// TIA Portal project "tictactoe_v2" (V14)

(* hardware
DEVICE "S7-1200 station_1"  S7-1200 Station
   slot 0: "Rack_0"  S7-1200 Rack  Rack  V1.0
   slot 1: "PLC_1"  CPU 1212C DC/DC/Rly  6ES7 212-1HE40-0XB0  V4.2
DEVICE "HMI_1"  KTP600 Basic color PN
   slot 0: "KTP600 Basic color PN"  KTP600 Basic color PN  6AV6 647-0AD11-3AX0  12.0.0.0
   slot 1: "HMI_RT_1"  KTP600 Basic color PN  6AV6 647-0AD11-3AX0  12.0.0.0
   slot 5: "HMI_1.IE_CP_1"  PROFINET Interface  12.0.0.0
      slot 1: "PROFINET Interface_1"  PROFINET Interface
         slot 1: "Port_1"  Port
*)

// ===== PLC "PLC_1"  CPU 1212C DC/DC/Rly =====

VAR_GLOBAL   // PLC tag table "Global"
   "x" AT %M15.2 : Bool;
   "Reset" AT %M12.1 : Bool;
   "GameType" AT %MB17 : SInt;
END_VAR

VAR_GLOBAL   // PLC tag table "3x3Tags"
   "t00" AT %MB1 : SInt;
   "t01" AT %MB2 : SInt;
   "t02" AT %MB3 : SInt;
   "t10" AT %MB4 : SInt;
   "t11" AT %MB10 : SInt;
   "t12" AT %MB13 : SInt;
   "t20" AT %MB7 : SInt;
   "t21" AT %MB8 : SInt;
   "t22" AT %MB9 : SInt;
   "t00btn" AT %M5.1 : Bool;
   "t01btn" AT %M5.2 : Bool;
   "t02btn" AT %M5.3 : Bool;
   "t10btn" AT %M5.4 : Bool;
   "t11btn" AT %M5.5 : Bool;
   "t12btn" AT %M5.6 : Bool;
   "t20btn" AT %M5.7 : Bool;
   "t21btn" AT %M6.0 : Bool;
   "t22btn" AT %M6.1 : Bool;
   "WinValue" AT %MB36 : SInt;
   "Stop" AT %M37.0 : Bool;
   "BotsTurn" AT %M37.1 : Bool;
   "t03" AT %MB46 : SInt;
   "t13" AT %MB38 : SInt;
   "t23" AT %MB39 : SInt;
   "t33" AT %MB40 : SInt;
   "t32" AT %MB41 : SInt;
   "t31" AT %MB42 : SInt;
   "t30" AT %MB43 : SInt;
   "t03btn" AT %M44.0 : Bool;
   "t13btn" AT %M44.1 : Bool;
   "t23btn" AT %M44.2 : Bool;
   "t33btn" AT %M44.3 : Bool;
   "t32btn" AT %M44.4 : Bool;
   "t31btn" AT %M44.5 : Bool;
   "t30btn" AT %M44.6 : Bool;
END_VAR

FUNCTION "ResetAllVariables" : Void   // FC1, LAD
{ S7_Optimized_Access := 'TRUE' }
VERSION : 0.1
BEGIN

REGION Network 1
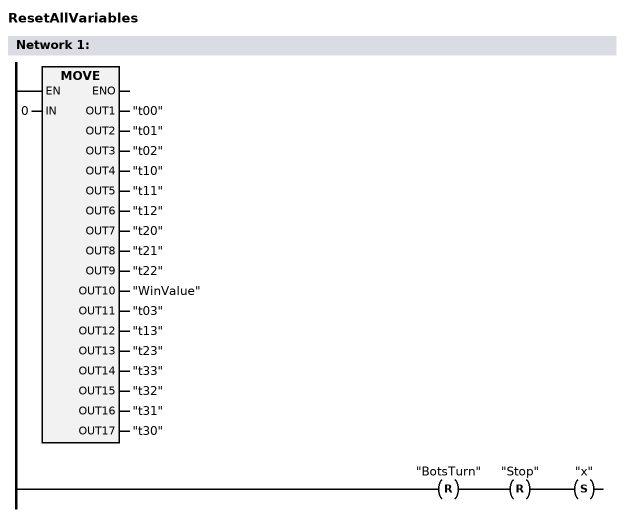
   RUNG wire#powerrail
      Move(in := 0, out1 => "t00", out2 => "t01", out3 => "t02", out4 => "t10", out5 => "t11", out6 => "t12", out7 => "t20", out8 => "t21", out9 => "t22", out10 => "WinValue", out11 => "t03", out12 => "t13", out13 => "t23", out14 => "t33", out15 => "t32", out16 => "t31", out17 => "t30")
   END_RUNG
   RUNG wire#powerrail
      R_Coil( "BotsTurn" )
      R_Coil( "Stop" )
      S_Coil( "x" )
   END_RUNG
   // the same network as SCL:
   "t00" := 0;
   "t01" := 0;
   "t02" := 0;
   "t10" := 0;
   "t11" := 0;
   "t12" := 0;
   "t20" := 0;
   "t21" := 0;
   "t22" := 0;
   "WinValue" := 0;
   "t03" := 0;
   "t13" := 0;
   "t23" := 0;
   "t33" := 0;
   "t32" := 0;
   "t31" := 0;
   "t30" := 0;
   "BotsTurn" := FALSE;
   "Stop" := FALSE;
   "x" := TRUE;
END_REGION
END_FUNCTION

FUNCTION "ChangeXValue" : Void   // FC4, LAD
{ S7_Optimized_Access := 'TRUE' }
VERSION : 0.1
   VAR_INPUT
      x : Bool;
   END_VAR
   VAR_OUTPUT
      value : Int;
   END_VAR
BEGIN

REGION Network 1
   // W zależności od wartości zmiennej "x" zmiana zapisywanego "symbolu"
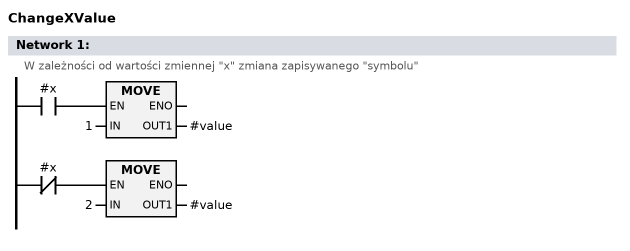
   RUNG wire#powerrail
      Contact( #x )
      Move(in := 1, out1 => #value)
   END_RUNG
   RUNG wire#powerrail
      I_Contact( #x )
      Move(in := 2, out1 => #value)
   END_RUNG
   // the same network as SCL:
   IF #x THEN #value := 1; END_IF;
   IF NOT #x THEN #value := 2; END_IF;
END_REGION
END_FUNCTION

ORGANIZATION_BLOCK "Main"   // OB1, LAD, ProgramCycle
TITLE = "Main Program Sweep (Cycle)"
{ S7_Optimized_Access := 'TRUE' }
VERSION : 0.1
   VAR_INPUT
      Initial_Call : Bool;   // Initial call of this OB
      Remanence : Bool;   // =True, if remanent data are available
   END_VAR
   VAR_TEMP
      temp : Bool;
      temp2 : Bool;
   END_VAR
BEGIN

REGION Network 1
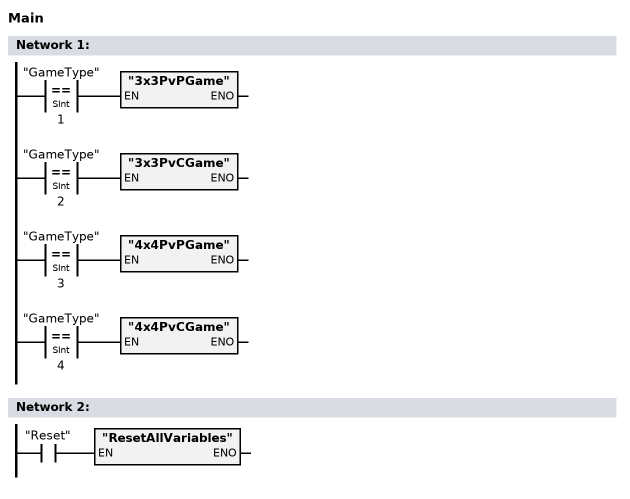
   RUNG wire#powerrail
      { S7_Templates := "SrcType := SInt" } EQ_Contact(in1 := "GameType", in2 := 1)
      "3x3PvPGame"()
   END_RUNG
   RUNG wire#powerrail
      { S7_Templates := "SrcType := SInt" } EQ_Contact(in1 := "GameType", in2 := 2)
      "3x3PvCGame"()
   END_RUNG
   RUNG wire#powerrail
      { S7_Templates := "SrcType := SInt" } EQ_Contact(in1 := "GameType", in2 := 3)
      "4x4PvPGame"()
   END_RUNG
   RUNG wire#powerrail
      { S7_Templates := "SrcType := SInt" } EQ_Contact(in1 := "GameType", in2 := 4)
      "4x4PvCGame"()
   END_RUNG
   // the same network as SCL:
   IF "GameType" = 1 THEN "3x3PvPGame"(); END_IF;
   IF "GameType" = 2 THEN "3x3PvCGame"(); END_IF;
   IF "GameType" = 3 THEN "4x4PvPGame"(); END_IF;
   IF "GameType" = 4 THEN "4x4PvCGame"(); END_IF;
END_REGION

REGION Network 2
   RUNG wire#powerrail
      Contact( "Reset" )
      "ResetAllVariables"()
   END_RUNG
   // the same network as SCL:
   IF "Reset" THEN "ResetAllVariables"(); END_IF;
END_REGION
END_ORGANIZATION_BLOCK

// folder: 3x3

FUNCTION "Check3x3" : Void   // FC2, LAD
{ S7_Optimized_Access := 'TRUE' }
VERSION : 0.1
   VAR_OUTPUT
      Stop : Bool;
      WinValue : SInt;
   END_VAR
BEGIN

REGION Network 1
   // Remis / X won!
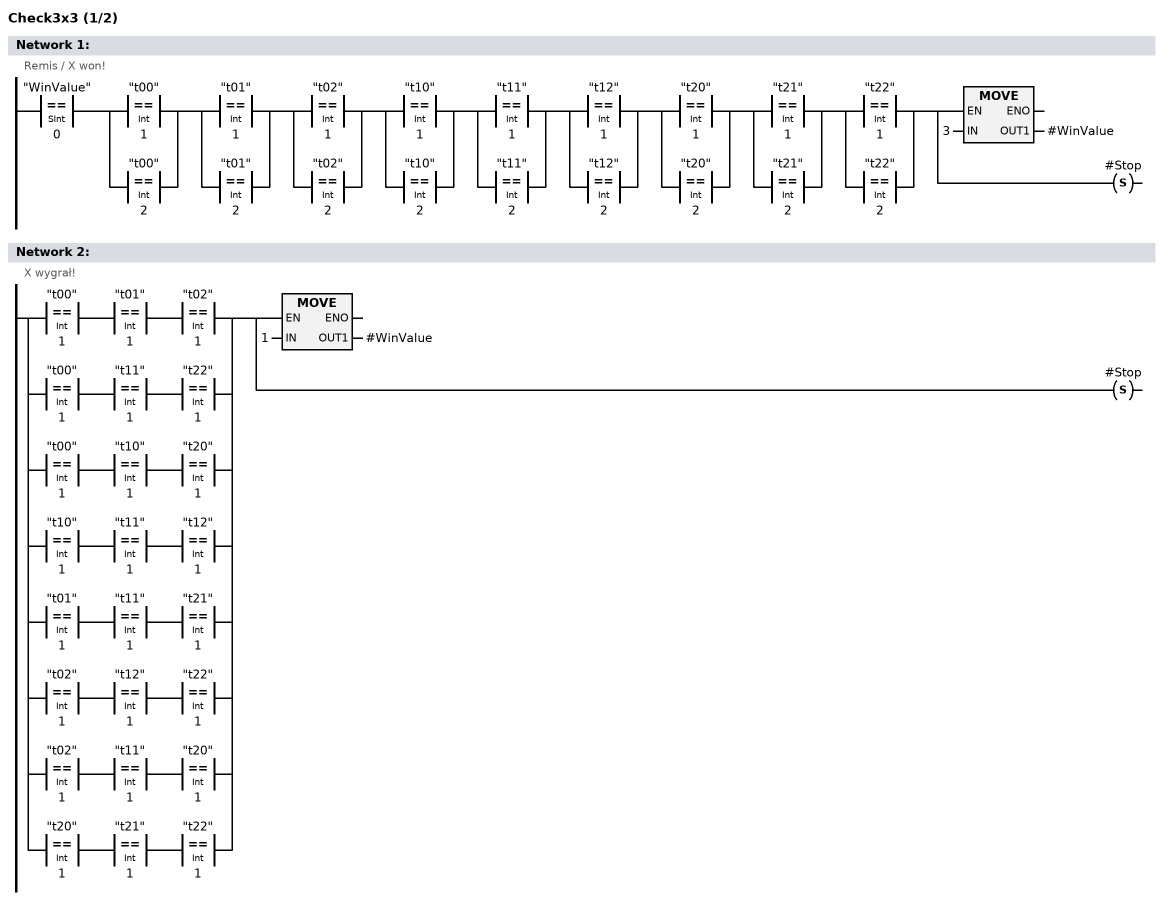
   RUNG wire#powerrail
      { S7_Templates := "SrcType := SInt" } EQ_Contact(in1 := "WinValue", in2 := 0)
      wire#w1
      { S7_Templates := "SrcType := Int" } EQ_Contact(in1 := "t00", in2 := 1)
      wire#w2
      { S7_Templates := "SrcType := Int" } EQ_Contact(in1 := "t01", in2 := 1)
      wire#w3
      { S7_Templates := "SrcType := Int" } EQ_Contact(in1 := "t02", in2 := 1)
      wire#w4
      { S7_Templates := "SrcType := Int" } EQ_Contact(in1 := "t10", in2 := 1)
      wire#w5
      { S7_Templates := "SrcType := Int" } EQ_Contact(in1 := "t11", in2 := 1)
      wire#w6
      { S7_Templates := "SrcType := Int" } EQ_Contact(in1 := "t12", in2 := 1)
      wire#w7
      { S7_Templates := "SrcType := Int" } EQ_Contact(in1 := "t20", in2 := 1)
      wire#w8
      { S7_Templates := "SrcType := Int" } EQ_Contact(in1 := "t21", in2 := 1)
      wire#w9
      { S7_Templates := "SrcType := Int" } EQ_Contact(in1 := "t22", in2 := 1)
      wire#w10
      Move(in := 3, out1 => #WinValue)
   END_RUNG
   RUNG wire#w1
      { S7_Templates := "SrcType := Int" } EQ_Contact(in1 := "t00", in2 := 2)
   END_RUNG wire#w2
   RUNG wire#w2
      { S7_Templates := "SrcType := Int" } EQ_Contact(in1 := "t01", in2 := 2)
   END_RUNG wire#w3
   RUNG wire#w3
      { S7_Templates := "SrcType := Int" } EQ_Contact(in1 := "t02", in2 := 2)
   END_RUNG wire#w4
   RUNG wire#w4
      { S7_Templates := "SrcType := Int" } EQ_Contact(in1 := "t10", in2 := 2)
   END_RUNG wire#w5
   RUNG wire#w5
      { S7_Templates := "SrcType := Int" } EQ_Contact(in1 := "t11", in2 := 2)
   END_RUNG wire#w6
   RUNG wire#w6
      { S7_Templates := "SrcType := Int" } EQ_Contact(in1 := "t12", in2 := 2)
   END_RUNG wire#w7
   RUNG wire#w7
      { S7_Templates := "SrcType := Int" } EQ_Contact(in1 := "t20", in2 := 2)
   END_RUNG wire#w8
   RUNG wire#w8
      { S7_Templates := "SrcType := Int" } EQ_Contact(in1 := "t21", in2 := 2)
   END_RUNG wire#w9
   RUNG wire#w9
      { S7_Templates := "SrcType := Int" } EQ_Contact(in1 := "t22", in2 := 2)
   END_RUNG wire#w10
   RUNG wire#w10
      S_Coil( #Stop )
   END_RUNG
   // the same network as SCL:
   IF ("WinValue" = 0) AND (("t00" = 1) OR ("t00" = 2)) AND (("t01" = 1) OR ("t01" = 2)) AND (("t02" = 1) OR ("t02" = 2)) AND (("t10" = 1) OR ("t10" = 2)) AND (("t11" = 1) OR ("t11" = 2)) AND (("t12" = 1) OR ("t12" = 2)) AND (("t20" = 1) OR ("t20" = 2)) AND (("t21" = 1) OR ("t21" = 2)) AND (("t22" = 1) OR ("t22" = 2)) THEN
       #WinValue := 3;
       #Stop := TRUE;
   END_IF;
END_REGION

REGION Network 2
   // X wygrał!
   RUNG wire#powerrail
      { S7_Templates := "SrcType := Int" } EQ_Contact(in1 := "t00", in2 := 1)
      { S7_Templates := "SrcType := Int" } EQ_Contact(in1 := "t01", in2 := 1)
      { S7_Templates := "SrcType := Int" } EQ_Contact(in1 := "t02", in2 := 1)
      wire#w1
      Move(in := 1, out1 => #WinValue)
   END_RUNG
   RUNG wire#powerrail
      { S7_Templates := "SrcType := Int" } EQ_Contact(in1 := "t00", in2 := 1)
      { S7_Templates := "SrcType := Int" } EQ_Contact(in1 := "t11", in2 := 1)
      { S7_Templates := "SrcType := Int" } EQ_Contact(in1 := "t22", in2 := 1)
   END_RUNG wire#w1
   RUNG wire#powerrail
      { S7_Templates := "SrcType := Int" } EQ_Contact(in1 := "t00", in2 := 1)
      { S7_Templates := "SrcType := Int" } EQ_Contact(in1 := "t10", in2 := 1)
      { S7_Templates := "SrcType := Int" } EQ_Contact(in1 := "t20", in2 := 1)
   END_RUNG wire#w1
   RUNG wire#powerrail
      { S7_Templates := "SrcType := Int" } EQ_Contact(in1 := "t10", in2 := 1)
      { S7_Templates := "SrcType := Int" } EQ_Contact(in1 := "t11", in2 := 1)
      { S7_Templates := "SrcType := Int" } EQ_Contact(in1 := "t12", in2 := 1)
   END_RUNG wire#w1
   RUNG wire#powerrail
      { S7_Templates := "SrcType := Int" } EQ_Contact(in1 := "t01", in2 := 1)
      { S7_Templates := "SrcType := Int" } EQ_Contact(in1 := "t11", in2 := 1)
      { S7_Templates := "SrcType := Int" } EQ_Contact(in1 := "t21", in2 := 1)
   END_RUNG wire#w1
   RUNG wire#powerrail
      { S7_Templates := "SrcType := Int" } EQ_Contact(in1 := "t02", in2 := 1)
      { S7_Templates := "SrcType := Int" } EQ_Contact(in1 := "t12", in2 := 1)
      { S7_Templates := "SrcType := Int" } EQ_Contact(in1 := "t22", in2 := 1)
   END_RUNG wire#w1
   RUNG wire#powerrail
      { S7_Templates := "SrcType := Int" } EQ_Contact(in1 := "t02", in2 := 1)
      { S7_Templates := "SrcType := Int" } EQ_Contact(in1 := "t11", in2 := 1)
      { S7_Templates := "SrcType := Int" } EQ_Contact(in1 := "t20", in2 := 1)
   END_RUNG wire#w1
   RUNG wire#powerrail
      { S7_Templates := "SrcType := Int" } EQ_Contact(in1 := "t20", in2 := 1)
      { S7_Templates := "SrcType := Int" } EQ_Contact(in1 := "t21", in2 := 1)
      { S7_Templates := "SrcType := Int" } EQ_Contact(in1 := "t22", in2 := 1)
   END_RUNG wire#w1
   RUNG wire#w1
      S_Coil( #Stop )
   END_RUNG
   // the same network as SCL:
   IF (("t00" = 1) AND ("t01" = 1) AND ("t02" = 1)) OR (("t00" = 1) AND ("t11" = 1) AND ("t22" = 1)) OR (("t00" = 1) AND ("t10" = 1) AND ("t20" = 1)) OR (("t10" = 1) AND ("t11" = 1) AND ("t12" = 1)) OR (("t01" = 1) AND ("t11" = 1) AND ("t21" = 1)) OR (("t02" = 1) AND ("t12" = 1) AND ("t22" = 1)) OR (("t02" = 1) AND ("t11" = 1) AND ("t20" = 1)) OR (("t20" = 1) AND ("t21" = 1) AND ("t22" = 1)) THEN
       #WinValue := 1;
       #Stop := TRUE;
   END_IF;
END_REGION

REGION Network 3
   // O wygrało! / O won! / O gewonnen!
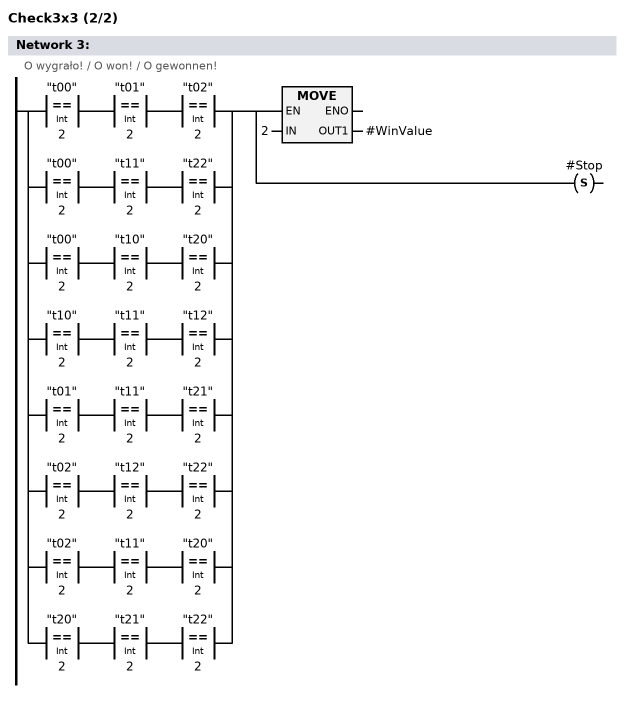
   RUNG wire#powerrail
      { S7_Templates := "SrcType := Int" } EQ_Contact(in1 := "t00", in2 := 2)
      { S7_Templates := "SrcType := Int" } EQ_Contact(in1 := "t01", in2 := 2)
      { S7_Templates := "SrcType := Int" } EQ_Contact(in1 := "t02", in2 := 2)
      wire#w1
      Move(in := 2, out1 => #WinValue)
   END_RUNG
   RUNG wire#powerrail
      { S7_Templates := "SrcType := Int" } EQ_Contact(in1 := "t00", in2 := 2)
      { S7_Templates := "SrcType := Int" } EQ_Contact(in1 := "t11", in2 := 2)
      { S7_Templates := "SrcType := Int" } EQ_Contact(in1 := "t22", in2 := 2)
   END_RUNG wire#w1
   RUNG wire#powerrail
      { S7_Templates := "SrcType := Int" } EQ_Contact(in1 := "t00", in2 := 2)
      { S7_Templates := "SrcType := Int" } EQ_Contact(in1 := "t10", in2 := 2)
      { S7_Templates := "SrcType := Int" } EQ_Contact(in1 := "t20", in2 := 2)
   END_RUNG wire#w1
   RUNG wire#powerrail
      { S7_Templates := "SrcType := Int" } EQ_Contact(in1 := "t10", in2 := 2)
      { S7_Templates := "SrcType := Int" } EQ_Contact(in1 := "t11", in2 := 2)
      { S7_Templates := "SrcType := Int" } EQ_Contact(in1 := "t12", in2 := 2)
   END_RUNG wire#w1
   RUNG wire#powerrail
      { S7_Templates := "SrcType := Int" } EQ_Contact(in1 := "t01", in2 := 2)
      { S7_Templates := "SrcType := Int" } EQ_Contact(in1 := "t11", in2 := 2)
      { S7_Templates := "SrcType := Int" } EQ_Contact(in1 := "t21", in2 := 2)
   END_RUNG wire#w1
   RUNG wire#powerrail
      { S7_Templates := "SrcType := Int" } EQ_Contact(in1 := "t02", in2 := 2)
      { S7_Templates := "SrcType := Int" } EQ_Contact(in1 := "t12", in2 := 2)
      { S7_Templates := "SrcType := Int" } EQ_Contact(in1 := "t22", in2 := 2)
   END_RUNG wire#w1
   RUNG wire#powerrail
      { S7_Templates := "SrcType := Int" } EQ_Contact(in1 := "t02", in2 := 2)
      { S7_Templates := "SrcType := Int" } EQ_Contact(in1 := "t11", in2 := 2)
      { S7_Templates := "SrcType := Int" } EQ_Contact(in1 := "t20", in2 := 2)
   END_RUNG wire#w1
   RUNG wire#powerrail
      { S7_Templates := "SrcType := Int" } EQ_Contact(in1 := "t20", in2 := 2)
      { S7_Templates := "SrcType := Int" } EQ_Contact(in1 := "t21", in2 := 2)
      { S7_Templates := "SrcType := Int" } EQ_Contact(in1 := "t22", in2 := 2)
   END_RUNG wire#w1
   RUNG wire#w1
      S_Coil( #Stop )
   END_RUNG
   // the same network as SCL:
   IF (("t00" = 2) AND ("t01" = 2) AND ("t02" = 2)) OR (("t00" = 2) AND ("t11" = 2) AND ("t22" = 2)) OR (("t00" = 2) AND ("t10" = 2) AND ("t20" = 2)) OR (("t10" = 2) AND ("t11" = 2) AND ("t12" = 2)) OR (("t01" = 2) AND ("t11" = 2) AND ("t21" = 2)) OR (("t02" = 2) AND ("t12" = 2) AND ("t22" = 2)) OR (("t02" = 2) AND ("t11" = 2) AND ("t20" = 2)) OR (("t20" = 2) AND ("t21" = 2) AND ("t22" = 2)) THEN
       #WinValue := 2;
       #Stop := TRUE;
   END_IF;
END_REGION

REGION Network 4
   // Remis
END_REGION
END_FUNCTION

// folder: 3x3/3x3PvC

FUNCTION "3x3PvCGame" : Void   // FC5, LAD
{ S7_Optimized_Access := 'TRUE' }
VERSION : 0.1
   VAR_TEMP
      temp00 : Bool;
      temp01 : Bool;
      temp02 : Bool;
      temp10 : Bool;
      temp11 : Bool;
      temp12 : Bool;
      temp20 : Bool;
      temp21 : Bool;
      temp22 : Bool;
      WINX : Bool;
      WINO : Bool;
      rngValue : Int;
      tempplayer : Bool;
      tempBot : Bool;
      tempMove : Bool;
   END_VAR
   VAR_TEMP   // added for the SCL form of the ladder/FBD networks
      _w1 : Bool;
      _w2 : Bool;
      _w3 : Bool;
      _w4 : Bool;
      _w5 : Bool;
      _w6 : Bool;
      _w7 : Bool;
      _w8 : Bool;
      _w9 : Bool;
      _w10 : Bool;
   END_VAR
BEGIN

REGION Network 1
   // Ruch gracza
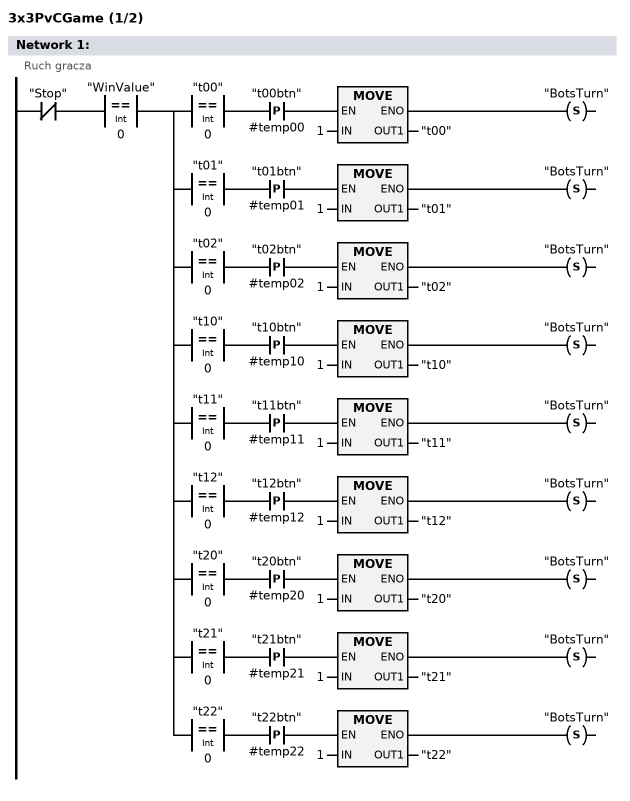
   RUNG wire#powerrail
      I_Contact( "Stop" )
      { S7_Templates := "SrcType := Int" } EQ_Contact(in1 := "WinValue", in2 := 0)
      wire#w1
      { S7_Templates := "SrcType := Int" } EQ_Contact(in1 := "t00", in2 := 0)
      P_Contact(operand := "t00btn", bit := #temp00)
      Move(in := 1, out1 => "t00")
      S_Coil( "BotsTurn" )
   END_RUNG
   RUNG wire#w1
      { S7_Templates := "SrcType := Int" } EQ_Contact(in1 := "t01", in2 := 0)
      P_Contact(operand := "t01btn", bit := #temp01)
      Move(in := 1, out1 => "t01")
      S_Coil( "BotsTurn" )
   END_RUNG
   RUNG wire#w1
      { S7_Templates := "SrcType := Int" } EQ_Contact(in1 := "t02", in2 := 0)
      P_Contact(operand := "t02btn", bit := #temp02)
      Move(in := 1, out1 => "t02")
      S_Coil( "BotsTurn" )
   END_RUNG
   RUNG wire#w1
      { S7_Templates := "SrcType := Int" } EQ_Contact(in1 := "t10", in2 := 0)
      P_Contact(operand := "t10btn", bit := #temp10)
      Move(in := 1, out1 => "t10")
      S_Coil( "BotsTurn" )
   END_RUNG
   RUNG wire#w1
      { S7_Templates := "SrcType := Int" } EQ_Contact(in1 := "t11", in2 := 0)
      P_Contact(operand := "t11btn", bit := #temp11)
      Move(in := 1, out1 => "t11")
      S_Coil( "BotsTurn" )
   END_RUNG
   RUNG wire#w1
      { S7_Templates := "SrcType := Int" } EQ_Contact(in1 := "t12", in2 := 0)
      P_Contact(operand := "t12btn", bit := #temp12)
      Move(in := 1, out1 => "t12")
      S_Coil( "BotsTurn" )
   END_RUNG
   RUNG wire#w1
      { S7_Templates := "SrcType := Int" } EQ_Contact(in1 := "t20", in2 := 0)
      P_Contact(operand := "t20btn", bit := #temp20)
      Move(in := 1, out1 => "t20")
      S_Coil( "BotsTurn" )
   END_RUNG
   RUNG wire#w1
      { S7_Templates := "SrcType := Int" } EQ_Contact(in1 := "t21", in2 := 0)
      P_Contact(operand := "t21btn", bit := #temp21)
      Move(in := 1, out1 => "t21")
      S_Coil( "BotsTurn" )
   END_RUNG
   RUNG wire#w1
      { S7_Templates := "SrcType := Int" } EQ_Contact(in1 := "t22", in2 := 0)
      P_Contact(operand := "t22btn", bit := #temp22)
      Move(in := 1, out1 => "t22")
      S_Coil( "BotsTurn" )
   END_RUNG
   // the same network as SCL:
   #_w1 := NOT "Stop" AND ("WinValue" = 0);
   #_w2 := #_w1 AND ("t00" = 0) AND "t00btn" AND NOT #temp00;   // rising edge of "t00btn"
   #temp00 := "t00btn";
   IF #_w2 THEN
       "t00" := 1;
       "BotsTurn" := TRUE;
   END_IF;
   #_w3 := #_w1 AND ("t01" = 0) AND "t01btn" AND NOT #temp01;   // rising edge of "t01btn"
   #temp01 := "t01btn";
   IF #_w3 THEN
       "t01" := 1;
       "BotsTurn" := TRUE;
   END_IF;
   #_w4 := #_w1 AND ("t02" = 0) AND "t02btn" AND NOT #temp02;   // rising edge of "t02btn"
   #temp02 := "t02btn";
   IF #_w4 THEN
       "t02" := 1;
       "BotsTurn" := TRUE;
   END_IF;
   #_w5 := #_w1 AND ("t10" = 0) AND "t10btn" AND NOT #temp10;   // rising edge of "t10btn"
   #temp10 := "t10btn";
   IF #_w5 THEN
       "t10" := 1;
       "BotsTurn" := TRUE;
   END_IF;
   #_w6 := #_w1 AND ("t11" = 0) AND "t11btn" AND NOT #temp11;   // rising edge of "t11btn"
   #temp11 := "t11btn";
   IF #_w6 THEN
       "t11" := 1;
       "BotsTurn" := TRUE;
   END_IF;
   #_w7 := #_w1 AND ("t12" = 0) AND "t12btn" AND NOT #temp12;   // rising edge of "t12btn"
   #temp12 := "t12btn";
   IF #_w7 THEN
       "t12" := 1;
       "BotsTurn" := TRUE;
   END_IF;
   #_w8 := #_w1 AND ("t20" = 0) AND "t20btn" AND NOT #temp20;   // rising edge of "t20btn"
   #temp20 := "t20btn";
   IF #_w8 THEN
       "t20" := 1;
       "BotsTurn" := TRUE;
   END_IF;
   #_w9 := #_w1 AND ("t21" = 0) AND "t21btn" AND NOT #temp21;   // rising edge of "t21btn"
   #temp21 := "t21btn";
   IF #_w9 THEN
       "t21" := 1;
       "BotsTurn" := TRUE;
   END_IF;
   #_w10 := #_w1 AND ("t22" = 0) AND "t22btn" AND NOT #temp22;   // rising edge of "t22btn"
   #temp22 := "t22btn";
   IF #_w10 THEN
       "t22" := 1;
       "BotsTurn" := TRUE;
   END_IF;
END_REGION

REGION Network 2
   // Ruch komputera
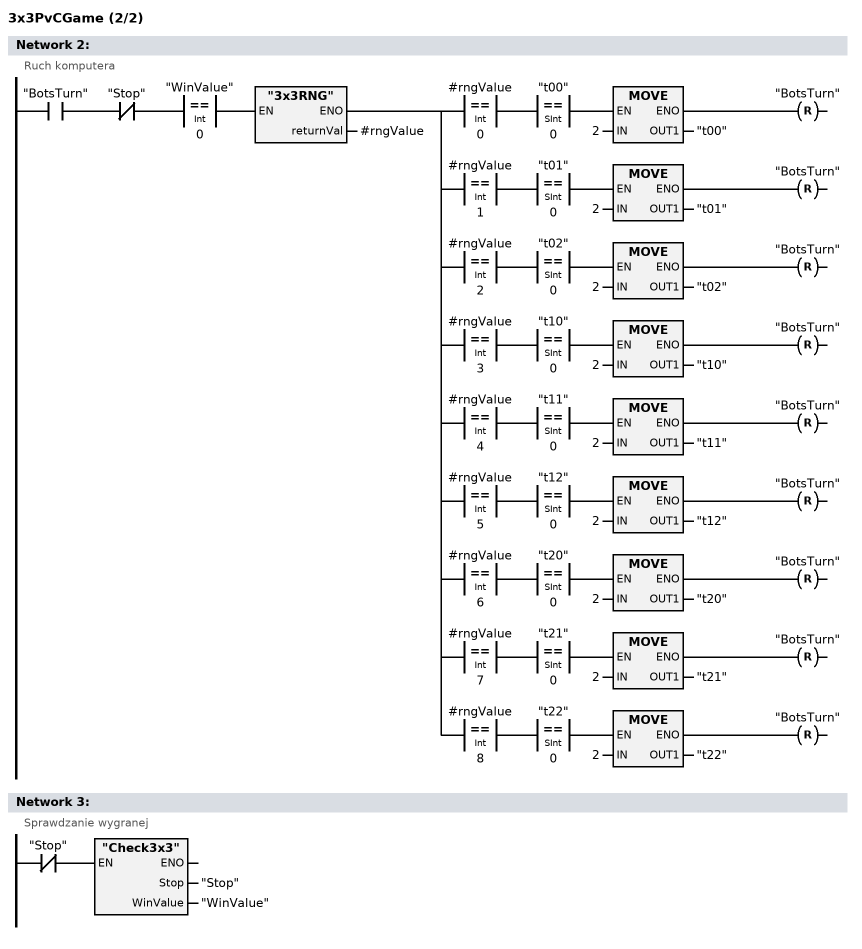
   RUNG wire#powerrail
      Contact( "BotsTurn" )
      I_Contact( "Stop" )
      { S7_Templates := "SrcType := Int" } EQ_Contact(in1 := "WinValue", in2 := 0)
      "3x3RNG"(returnVal => #rngValue)
      wire#w1
      { S7_Templates := "SrcType := Int" } EQ_Contact(in1 := #rngValue, in2 := 0)
      { S7_Templates := "SrcType := SInt" } EQ_Contact(in1 := "t00", in2 := 0)
      Move(in := 2, out1 => "t00")
      R_Coil( "BotsTurn" )
   END_RUNG
   RUNG wire#w1
      { S7_Templates := "SrcType := Int" } EQ_Contact(in1 := #rngValue, in2 := 1)
      { S7_Templates := "SrcType := SInt" } EQ_Contact(in1 := "t01", in2 := 0)
      Move(in := 2, out1 => "t01")
      R_Coil( "BotsTurn" )
   END_RUNG
   RUNG wire#w1
      { S7_Templates := "SrcType := Int" } EQ_Contact(in1 := #rngValue, in2 := 2)
      { S7_Templates := "SrcType := SInt" } EQ_Contact(in1 := "t02", in2 := 0)
      Move(in := 2, out1 => "t02")
      R_Coil( "BotsTurn" )
   END_RUNG
   RUNG wire#w1
      { S7_Templates := "SrcType := Int" } EQ_Contact(in1 := #rngValue, in2 := 3)
      { S7_Templates := "SrcType := SInt" } EQ_Contact(in1 := "t10", in2 := 0)
      Move(in := 2, out1 => "t10")
      R_Coil( "BotsTurn" )
   END_RUNG
   RUNG wire#w1
      { S7_Templates := "SrcType := Int" } EQ_Contact(in1 := #rngValue, in2 := 4)
      { S7_Templates := "SrcType := SInt" } EQ_Contact(in1 := "t11", in2 := 0)
      Move(in := 2, out1 => "t11")
      R_Coil( "BotsTurn" )
   END_RUNG
   RUNG wire#w1
      { S7_Templates := "SrcType := Int" } EQ_Contact(in1 := #rngValue, in2 := 5)
      { S7_Templates := "SrcType := SInt" } EQ_Contact(in1 := "t12", in2 := 0)
      Move(in := 2, out1 => "t12")
      R_Coil( "BotsTurn" )
   END_RUNG
   RUNG wire#w1
      { S7_Templates := "SrcType := Int" } EQ_Contact(in1 := #rngValue, in2 := 6)
      { S7_Templates := "SrcType := SInt" } EQ_Contact(in1 := "t20", in2 := 0)
      Move(in := 2, out1 => "t20")
      R_Coil( "BotsTurn" )
   END_RUNG
   RUNG wire#w1
      { S7_Templates := "SrcType := Int" } EQ_Contact(in1 := #rngValue, in2 := 7)
      { S7_Templates := "SrcType := SInt" } EQ_Contact(in1 := "t21", in2 := 0)
      Move(in := 2, out1 => "t21")
      R_Coil( "BotsTurn" )
   END_RUNG
   RUNG wire#w1
      { S7_Templates := "SrcType := Int" } EQ_Contact(in1 := #rngValue, in2 := 8)
      { S7_Templates := "SrcType := SInt" } EQ_Contact(in1 := "t22", in2 := 0)
      Move(in := 2, out1 => "t22")
      R_Coil( "BotsTurn" )
   END_RUNG
   // the same network as SCL:
   "3x3RNG"(EN := "BotsTurn" AND NOT "Stop" AND ("WinValue" = 0), returnVal => #rngValue, ENO => #_w1);
   #_w2 := #_w1 AND (#rngValue = 0) AND ("t00" = 0);
   IF #_w2 THEN
       "t00" := 2;
       "BotsTurn" := FALSE;
   END_IF;
   #_w3 := #_w1 AND (#rngValue = 1) AND ("t01" = 0);
   IF #_w3 THEN
       "t01" := 2;
       "BotsTurn" := FALSE;
   END_IF;
   #_w4 := #_w1 AND (#rngValue = 2) AND ("t02" = 0);
   IF #_w4 THEN
       "t02" := 2;
       "BotsTurn" := FALSE;
   END_IF;
   #_w5 := #_w1 AND (#rngValue = 3) AND ("t10" = 0);
   IF #_w5 THEN
       "t10" := 2;
       "BotsTurn" := FALSE;
   END_IF;
   #_w6 := #_w1 AND (#rngValue = 4) AND ("t11" = 0);
   IF #_w6 THEN
       "t11" := 2;
       "BotsTurn" := FALSE;
   END_IF;
   #_w7 := #_w1 AND (#rngValue = 5) AND ("t12" = 0);
   IF #_w7 THEN
       "t12" := 2;
       "BotsTurn" := FALSE;
   END_IF;
   #_w8 := #_w1 AND (#rngValue = 6) AND ("t20" = 0);
   IF #_w8 THEN
       "t20" := 2;
       "BotsTurn" := FALSE;
   END_IF;
   #_w9 := #_w1 AND (#rngValue = 7) AND ("t21" = 0);
   IF #_w9 THEN
       "t21" := 2;
       "BotsTurn" := FALSE;
   END_IF;
   #_w10 := #_w1 AND (#rngValue = 8) AND ("t22" = 0);
   IF #_w10 THEN
       "t22" := 2;
       "BotsTurn" := FALSE;
   END_IF;
END_REGION

REGION Network 3
   // Sprawdzanie wygranej
   RUNG wire#powerrail
      I_Contact( "Stop" )
      "Check3x3"(Stop => "Stop", WinValue => "WinValue")
   END_RUNG
   // the same network as SCL:
   IF NOT "Stop" THEN "Check3x3"(Stop => "Stop", WinValue => "WinValue"); END_IF;
END_REGION
END_FUNCTION

FUNCTION "3x3RNG" : Void   // FC11, LAD
{ S7_Optimized_Access := 'TRUE' }
VERSION : 0.1
   VAR_OUTPUT
      returnVal : Int;
   END_VAR
   VAR_TEMP
      val : Int;
      reset : Bool;
      Stop : Bool;
      datetemp : DTL;
   END_VAR
BEGIN

REGION Network 1
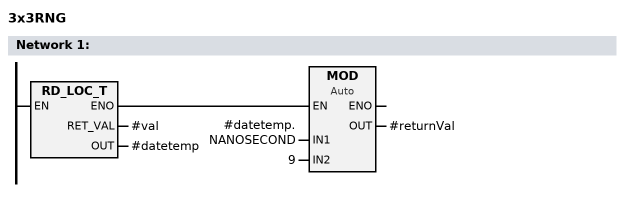
   // ENO of a box is taken as its EN; it also drops when the box reports an error
   #val := RD_LOC_T(OUT => #datetemp);
   #returnVal := #datetemp.NANOSECOND MOD 9;
END_REGION
END_FUNCTION

// folder: 3x3/3x3PvP

FUNCTION "3x3PvPGame" : Void   // FC3, LAD
{ S7_Optimized_Access := 'TRUE' }
VERSION : 0.1
   VAR_TEMP
      temp00 : Bool;
      temp01 : Bool;
      temp02 : Bool;
      temp10 : Bool;
      temp11 : Bool;
      temp12 : Bool;
      temp20 : Bool;
      temp21 : Bool;
      temp22 : Bool;
      WINX : Bool;
      WINO : Bool;
   END_VAR
   VAR_TEMP   // added for the SCL form of the ladder/FBD networks
      _w1 : Bool;
      _w2 : Bool;
      _w3 : Bool;
      _w4 : Bool;
      _w5 : Bool;
      _w6 : Bool;
      _w7 : Bool;
      _w8 : Bool;
      _w9 : Bool;
      _w10 : Bool;
   END_VAR
BEGIN

REGION Network 1
   // Ruch gracza - zmienny symbol
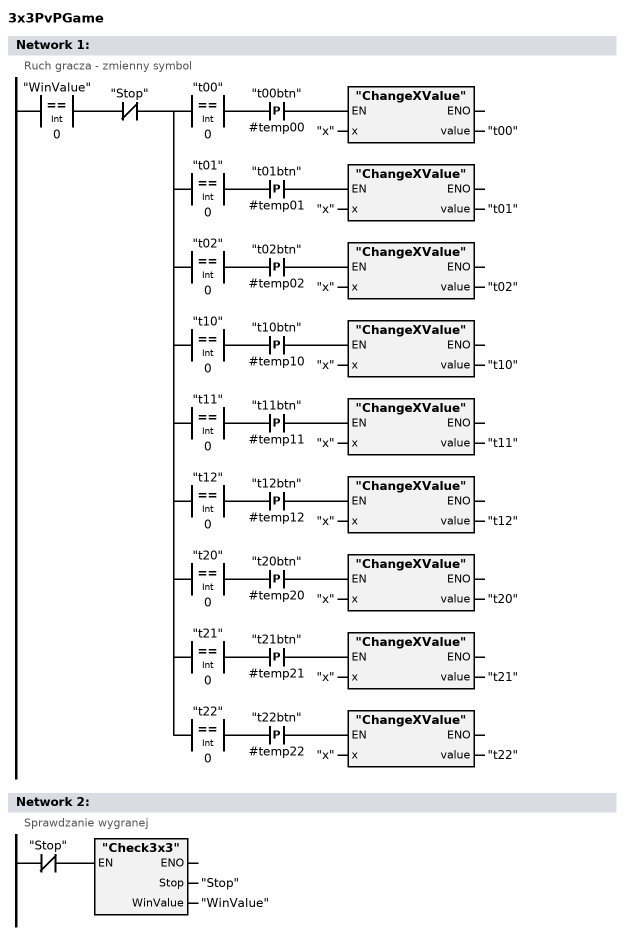
   RUNG wire#powerrail
      { S7_Templates := "SrcType := Int" } EQ_Contact(in1 := "WinValue", in2 := 0)
      I_Contact( "Stop" )
      wire#w1
      { S7_Templates := "SrcType := Int" } EQ_Contact(in1 := "t00", in2 := 0)
      P_Contact(operand := "t00btn", bit := #temp00)
      "ChangeXValue"(x := "x", value => "t00")
   END_RUNG
   RUNG wire#w1
      { S7_Templates := "SrcType := Int" } EQ_Contact(in1 := "t01", in2 := 0)
      P_Contact(operand := "t01btn", bit := #temp01)
      "ChangeXValue"(x := "x", value => "t01")
   END_RUNG
   RUNG wire#w1
      { S7_Templates := "SrcType := Int" } EQ_Contact(in1 := "t02", in2 := 0)
      P_Contact(operand := "t02btn", bit := #temp02)
      "ChangeXValue"(x := "x", value => "t02")
   END_RUNG
   RUNG wire#w1
      { S7_Templates := "SrcType := Int" } EQ_Contact(in1 := "t10", in2 := 0)
      P_Contact(operand := "t10btn", bit := #temp10)
      "ChangeXValue"(x := "x", value => "t10")
   END_RUNG
   RUNG wire#w1
      { S7_Templates := "SrcType := Int" } EQ_Contact(in1 := "t11", in2 := 0)
      P_Contact(operand := "t11btn", bit := #temp11)
      "ChangeXValue"(x := "x", value => "t11")
   END_RUNG
   RUNG wire#w1
      { S7_Templates := "SrcType := Int" } EQ_Contact(in1 := "t12", in2 := 0)
      P_Contact(operand := "t12btn", bit := #temp12)
      "ChangeXValue"(x := "x", value => "t12")
   END_RUNG
   RUNG wire#w1
      { S7_Templates := "SrcType := Int" } EQ_Contact(in1 := "t20", in2 := 0)
      P_Contact(operand := "t20btn", bit := #temp20)
      "ChangeXValue"(x := "x", value => "t20")
   END_RUNG
   RUNG wire#w1
      { S7_Templates := "SrcType := Int" } EQ_Contact(in1 := "t21", in2 := 0)
      P_Contact(operand := "t21btn", bit := #temp21)
      "ChangeXValue"(x := "x", value => "t21")
   END_RUNG
   RUNG wire#w1
      { S7_Templates := "SrcType := Int" } EQ_Contact(in1 := "t22", in2 := 0)
      P_Contact(operand := "t22btn", bit := #temp22)
      "ChangeXValue"(x := "x", value => "t22")
   END_RUNG
   // the same network as SCL:
   #_w1 := ("WinValue" = 0) AND NOT "Stop";
   #_w2 := #_w1 AND ("t00" = 0) AND "t00btn" AND NOT #temp00;   // rising edge of "t00btn"
   #temp00 := "t00btn";
   IF #_w2 THEN "ChangeXValue"(x := "x", value => "t00"); END_IF;
   #_w3 := #_w1 AND ("t01" = 0) AND "t01btn" AND NOT #temp01;   // rising edge of "t01btn"
   #temp01 := "t01btn";
   IF #_w3 THEN "ChangeXValue"(x := "x", value => "t01"); END_IF;
   #_w4 := #_w1 AND ("t02" = 0) AND "t02btn" AND NOT #temp02;   // rising edge of "t02btn"
   #temp02 := "t02btn";
   IF #_w4 THEN "ChangeXValue"(x := "x", value => "t02"); END_IF;
   #_w5 := #_w1 AND ("t10" = 0) AND "t10btn" AND NOT #temp10;   // rising edge of "t10btn"
   #temp10 := "t10btn";
   IF #_w5 THEN "ChangeXValue"(x := "x", value => "t10"); END_IF;
   #_w6 := #_w1 AND ("t11" = 0) AND "t11btn" AND NOT #temp11;   // rising edge of "t11btn"
   #temp11 := "t11btn";
   IF #_w6 THEN "ChangeXValue"(x := "x", value => "t11"); END_IF;
   #_w7 := #_w1 AND ("t12" = 0) AND "t12btn" AND NOT #temp12;   // rising edge of "t12btn"
   #temp12 := "t12btn";
   IF #_w7 THEN "ChangeXValue"(x := "x", value => "t12"); END_IF;
   #_w8 := #_w1 AND ("t20" = 0) AND "t20btn" AND NOT #temp20;   // rising edge of "t20btn"
   #temp20 := "t20btn";
   IF #_w8 THEN "ChangeXValue"(x := "x", value => "t20"); END_IF;
   #_w9 := #_w1 AND ("t21" = 0) AND "t21btn" AND NOT #temp21;   // rising edge of "t21btn"
   #temp21 := "t21btn";
   IF #_w9 THEN "ChangeXValue"(x := "x", value => "t21"); END_IF;
   #_w10 := #_w1 AND ("t22" = 0) AND "t22btn" AND NOT #temp22;   // rising edge of "t22btn"
   #temp22 := "t22btn";
   IF #_w10 THEN "ChangeXValue"(x := "x", value => "t22"); END_IF;
END_REGION

REGION Network 2
   // Sprawdzanie wygranej
   RUNG wire#powerrail
      I_Contact( "Stop" )
      "Check3x3"(Stop => "Stop", WinValue => "WinValue")
   END_RUNG
   // the same network as SCL:
   IF NOT "Stop" THEN "Check3x3"(Stop => "Stop", WinValue => "WinValue"); END_IF;
END_REGION
END_FUNCTION

// folder: 4x4

FUNCTION "Check4x4" : Void   // FC8, LAD
{ S7_Optimized_Access := 'TRUE' }
VERSION : 0.1
   VAR_OUTPUT
      Stop : Bool;
      WinValue : SInt;
   END_VAR
BEGIN

REGION Network 1
   // Remis
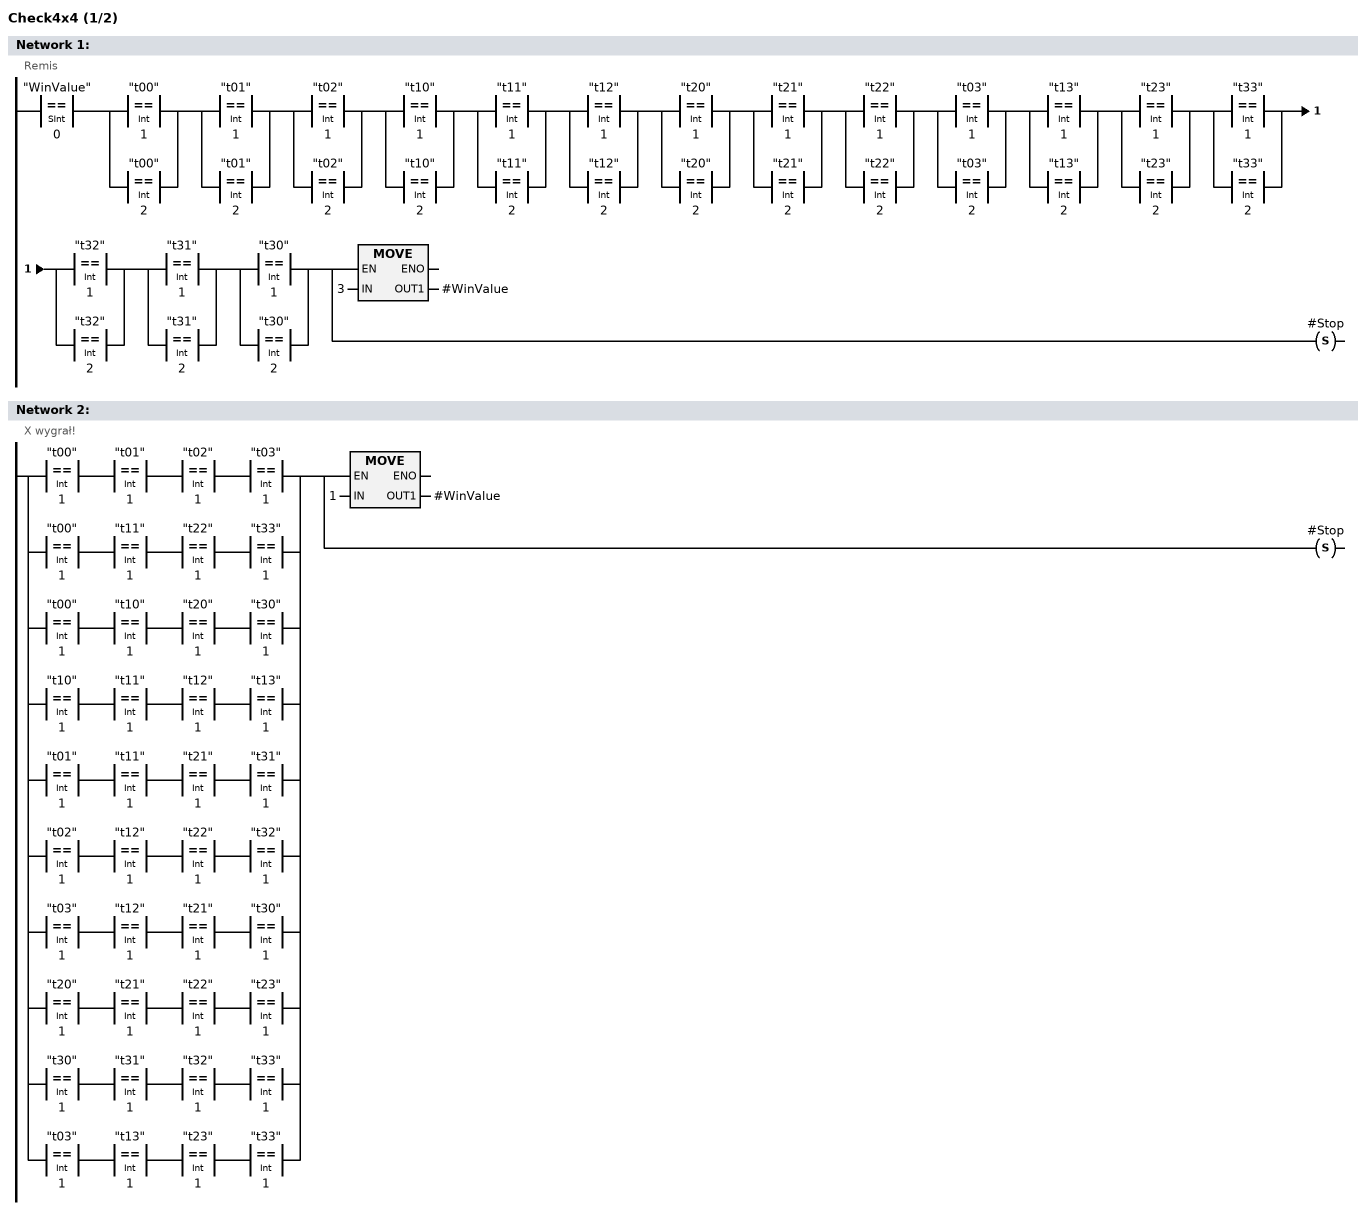
   RUNG wire#powerrail
      { S7_Templates := "SrcType := SInt" } EQ_Contact(in1 := "WinValue", in2 := 0)
      wire#w1
      { S7_Templates := "SrcType := Int" } EQ_Contact(in1 := "t00", in2 := 1)
      wire#w2
      { S7_Templates := "SrcType := Int" } EQ_Contact(in1 := "t01", in2 := 1)
      wire#w3
      { S7_Templates := "SrcType := Int" } EQ_Contact(in1 := "t02", in2 := 1)
      wire#w4
      { S7_Templates := "SrcType := Int" } EQ_Contact(in1 := "t10", in2 := 1)
      wire#w5
      { S7_Templates := "SrcType := Int" } EQ_Contact(in1 := "t11", in2 := 1)
      wire#w6
      { S7_Templates := "SrcType := Int" } EQ_Contact(in1 := "t12", in2 := 1)
      wire#w7
      { S7_Templates := "SrcType := Int" } EQ_Contact(in1 := "t20", in2 := 1)
      wire#w8
      { S7_Templates := "SrcType := Int" } EQ_Contact(in1 := "t21", in2 := 1)
      wire#w9
      { S7_Templates := "SrcType := Int" } EQ_Contact(in1 := "t22", in2 := 1)
      wire#w10
      { S7_Templates := "SrcType := Int" } EQ_Contact(in1 := "t03", in2 := 1)
      wire#w11
      { S7_Templates := "SrcType := Int" } EQ_Contact(in1 := "t13", in2 := 1)
      wire#w12
      { S7_Templates := "SrcType := Int" } EQ_Contact(in1 := "t23", in2 := 1)
      wire#w13
      { S7_Templates := "SrcType := Int" } EQ_Contact(in1 := "t33", in2 := 1)
      wire#w14
      { S7_Templates := "SrcType := Int" } EQ_Contact(in1 := "t32", in2 := 1)
      wire#w15
      { S7_Templates := "SrcType := Int" } EQ_Contact(in1 := "t31", in2 := 1)
      wire#w16
      { S7_Templates := "SrcType := Int" } EQ_Contact(in1 := "t30", in2 := 1)
      wire#w17
      Move(in := 3, out1 => #WinValue)
   END_RUNG
   RUNG wire#w1
      { S7_Templates := "SrcType := Int" } EQ_Contact(in1 := "t00", in2 := 2)
   END_RUNG wire#w2
   RUNG wire#w2
      { S7_Templates := "SrcType := Int" } EQ_Contact(in1 := "t01", in2 := 2)
   END_RUNG wire#w3
   RUNG wire#w3
      { S7_Templates := "SrcType := Int" } EQ_Contact(in1 := "t02", in2 := 2)
   END_RUNG wire#w4
   RUNG wire#w4
      { S7_Templates := "SrcType := Int" } EQ_Contact(in1 := "t10", in2 := 2)
   END_RUNG wire#w5
   RUNG wire#w5
      { S7_Templates := "SrcType := Int" } EQ_Contact(in1 := "t11", in2 := 2)
   END_RUNG wire#w6
   RUNG wire#w6
      { S7_Templates := "SrcType := Int" } EQ_Contact(in1 := "t12", in2 := 2)
   END_RUNG wire#w7
   RUNG wire#w7
      { S7_Templates := "SrcType := Int" } EQ_Contact(in1 := "t20", in2 := 2)
   END_RUNG wire#w8
   RUNG wire#w8
      { S7_Templates := "SrcType := Int" } EQ_Contact(in1 := "t21", in2 := 2)
   END_RUNG wire#w9
   RUNG wire#w9
      { S7_Templates := "SrcType := Int" } EQ_Contact(in1 := "t22", in2 := 2)
   END_RUNG wire#w10
   RUNG wire#w10
      { S7_Templates := "SrcType := Int" } EQ_Contact(in1 := "t03", in2 := 2)
   END_RUNG wire#w11
   RUNG wire#w11
      { S7_Templates := "SrcType := Int" } EQ_Contact(in1 := "t13", in2 := 2)
   END_RUNG wire#w12
   RUNG wire#w12
      { S7_Templates := "SrcType := Int" } EQ_Contact(in1 := "t23", in2 := 2)
   END_RUNG wire#w13
   RUNG wire#w13
      { S7_Templates := "SrcType := Int" } EQ_Contact(in1 := "t33", in2 := 2)
   END_RUNG wire#w14
   RUNG wire#w14
      { S7_Templates := "SrcType := Int" } EQ_Contact(in1 := "t32", in2 := 2)
   END_RUNG wire#w15
   RUNG wire#w15
      { S7_Templates := "SrcType := Int" } EQ_Contact(in1 := "t31", in2 := 2)
   END_RUNG wire#w16
   RUNG wire#w16
      { S7_Templates := "SrcType := Int" } EQ_Contact(in1 := "t30", in2 := 2)
   END_RUNG wire#w17
   RUNG wire#w17
      S_Coil( #Stop )
   END_RUNG
   // the same network as SCL:
   IF ("WinValue" = 0) AND (("t00" = 1) OR ("t00" = 2)) AND (("t01" = 1) OR ("t01" = 2)) AND (("t02" = 1) OR ("t02" = 2)) AND (("t10" = 1) OR ("t10" = 2)) AND (("t11" = 1) OR ("t11" = 2)) AND (("t12" = 1) OR ("t12" = 2)) AND (("t20" = 1) OR ("t20" = 2)) AND (("t21" = 1) OR ("t21" = 2)) AND (("t22" = 1) OR ("t22" = 2)) AND (("t03" = 1) OR ("t03" = 2)) AND (("t13" = 1) OR ("t13" = 2)) AND (("t23" = 1) OR ("t23" = 2)) AND (("t33" = 1) OR ("t33" = 2)) AND (("t32" = 1) OR ("t32" = 2)) AND (("t31" = 1) OR ("t31" = 2)) AND (("t30" = 1) OR ("t30" = 2)) THEN
       #WinValue := 3;
       #Stop := TRUE;
   END_IF;
END_REGION

REGION Network 2
   // X wygrał!
   RUNG wire#powerrail
      { S7_Templates := "SrcType := Int" } EQ_Contact(in1 := "t00", in2 := 1)
      { S7_Templates := "SrcType := Int" } EQ_Contact(in1 := "t01", in2 := 1)
      { S7_Templates := "SrcType := Int" } EQ_Contact(in1 := "t02", in2 := 1)
      { S7_Templates := "SrcType := Int" } EQ_Contact(in1 := "t03", in2 := 1)
      wire#w1
      Move(in := 1, out1 => #WinValue)
   END_RUNG
   RUNG wire#powerrail
      { S7_Templates := "SrcType := Int" } EQ_Contact(in1 := "t00", in2 := 1)
      { S7_Templates := "SrcType := Int" } EQ_Contact(in1 := "t11", in2 := 1)
      { S7_Templates := "SrcType := Int" } EQ_Contact(in1 := "t22", in2 := 1)
      { S7_Templates := "SrcType := Int" } EQ_Contact(in1 := "t33", in2 := 1)
   END_RUNG wire#w1
   RUNG wire#powerrail
      { S7_Templates := "SrcType := Int" } EQ_Contact(in1 := "t00", in2 := 1)
      { S7_Templates := "SrcType := Int" } EQ_Contact(in1 := "t10", in2 := 1)
      { S7_Templates := "SrcType := Int" } EQ_Contact(in1 := "t20", in2 := 1)
      { S7_Templates := "SrcType := Int" } EQ_Contact(in1 := "t30", in2 := 1)
   END_RUNG wire#w1
   RUNG wire#powerrail
      { S7_Templates := "SrcType := Int" } EQ_Contact(in1 := "t10", in2 := 1)
      { S7_Templates := "SrcType := Int" } EQ_Contact(in1 := "t11", in2 := 1)
      { S7_Templates := "SrcType := Int" } EQ_Contact(in1 := "t12", in2 := 1)
      { S7_Templates := "SrcType := Int" } EQ_Contact(in1 := "t13", in2 := 1)
   END_RUNG wire#w1
   RUNG wire#powerrail
      { S7_Templates := "SrcType := Int" } EQ_Contact(in1 := "t01", in2 := 1)
      { S7_Templates := "SrcType := Int" } EQ_Contact(in1 := "t11", in2 := 1)
      { S7_Templates := "SrcType := Int" } EQ_Contact(in1 := "t21", in2 := 1)
      { S7_Templates := "SrcType := Int" } EQ_Contact(in1 := "t31", in2 := 1)
   END_RUNG wire#w1
   RUNG wire#powerrail
      { S7_Templates := "SrcType := Int" } EQ_Contact(in1 := "t02", in2 := 1)
      { S7_Templates := "SrcType := Int" } EQ_Contact(in1 := "t12", in2 := 1)
      { S7_Templates := "SrcType := Int" } EQ_Contact(in1 := "t22", in2 := 1)
      { S7_Templates := "SrcType := Int" } EQ_Contact(in1 := "t32", in2 := 1)
   END_RUNG wire#w1
   RUNG wire#powerrail
      { S7_Templates := "SrcType := Int" } EQ_Contact(in1 := "t03", in2 := 1)
      { S7_Templates := "SrcType := Int" } EQ_Contact(in1 := "t12", in2 := 1)
      { S7_Templates := "SrcType := Int" } EQ_Contact(in1 := "t21", in2 := 1)
      { S7_Templates := "SrcType := Int" } EQ_Contact(in1 := "t30", in2 := 1)
   END_RUNG wire#w1
   RUNG wire#powerrail
      { S7_Templates := "SrcType := Int" } EQ_Contact(in1 := "t20", in2 := 1)
      { S7_Templates := "SrcType := Int" } EQ_Contact(in1 := "t21", in2 := 1)
      { S7_Templates := "SrcType := Int" } EQ_Contact(in1 := "t22", in2 := 1)
      { S7_Templates := "SrcType := Int" } EQ_Contact(in1 := "t23", in2 := 1)
   END_RUNG wire#w1
   RUNG wire#powerrail
      { S7_Templates := "SrcType := Int" } EQ_Contact(in1 := "t30", in2 := 1)
      { S7_Templates := "SrcType := Int" } EQ_Contact(in1 := "t31", in2 := 1)
      { S7_Templates := "SrcType := Int" } EQ_Contact(in1 := "t32", in2 := 1)
      { S7_Templates := "SrcType := Int" } EQ_Contact(in1 := "t33", in2 := 1)
   END_RUNG wire#w1
   RUNG wire#powerrail
      { S7_Templates := "SrcType := Int" } EQ_Contact(in1 := "t03", in2 := 1)
      { S7_Templates := "SrcType := Int" } EQ_Contact(in1 := "t13", in2 := 1)
      { S7_Templates := "SrcType := Int" } EQ_Contact(in1 := "t23", in2 := 1)
      { S7_Templates := "SrcType := Int" } EQ_Contact(in1 := "t33", in2 := 1)
   END_RUNG wire#w1
   RUNG wire#w1
      S_Coil( #Stop )
   END_RUNG
   // the same network as SCL:
   IF (("t00" = 1) AND ("t01" = 1) AND ("t02" = 1) AND ("t03" = 1)) OR (("t00" = 1) AND ("t11" = 1) AND ("t22" = 1) AND ("t33" = 1)) OR (("t00" = 1) AND ("t10" = 1) AND ("t20" = 1) AND ("t30" = 1)) OR (("t10" = 1) AND ("t11" = 1) AND ("t12" = 1) AND ("t13" = 1)) OR (("t01" = 1) AND ("t11" = 1) AND ("t21" = 1) AND ("t31" = 1)) OR (("t02" = 1) AND ("t12" = 1) AND ("t22" = 1) AND ("t32" = 1)) OR (("t03" = 1) AND ("t12" = 1) AND ("t21" = 1) AND ("t30" = 1)) OR (("t20" = 1) AND ("t21" = 1) AND ("t22" = 1) AND ("t23" = 1)) OR (("t30" = 1) AND ("t31" = 1) AND ("t32" = 1) AND ("t33" = 1)) OR (("t03" = 1) AND ("t13" = 1) AND ("t23" = 1) AND ("t33" = 1)) THEN
       #WinValue := 1;
       #Stop := TRUE;
   END_IF;
END_REGION

REGION Network 3
   // O wygrało!
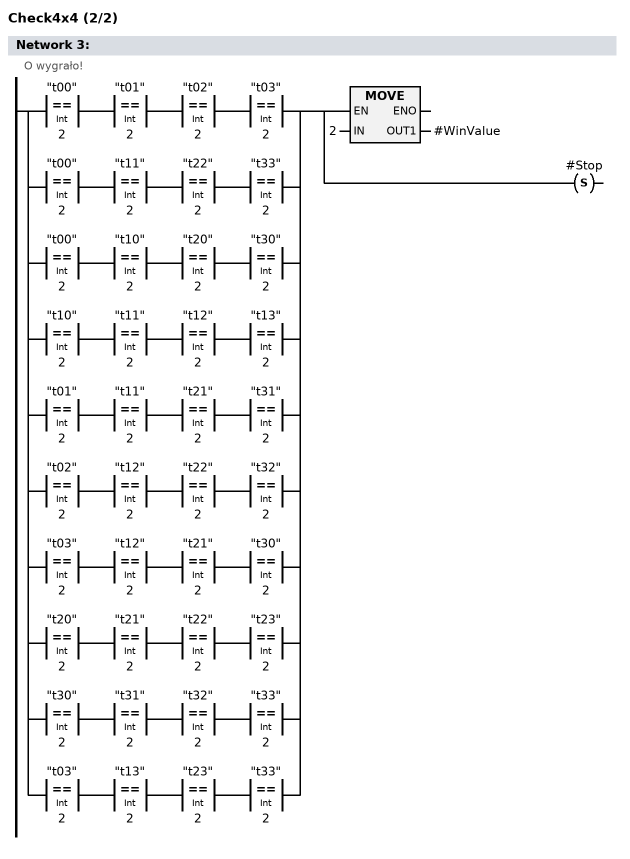
   RUNG wire#powerrail
      { S7_Templates := "SrcType := Int" } EQ_Contact(in1 := "t00", in2 := 2)
      { S7_Templates := "SrcType := Int" } EQ_Contact(in1 := "t01", in2 := 2)
      { S7_Templates := "SrcType := Int" } EQ_Contact(in1 := "t02", in2 := 2)
      { S7_Templates := "SrcType := Int" } EQ_Contact(in1 := "t03", in2 := 2)
      wire#w1
      Move(in := 2, out1 => #WinValue)
   END_RUNG
   RUNG wire#powerrail
      { S7_Templates := "SrcType := Int" } EQ_Contact(in1 := "t00", in2 := 2)
      { S7_Templates := "SrcType := Int" } EQ_Contact(in1 := "t11", in2 := 2)
      { S7_Templates := "SrcType := Int" } EQ_Contact(in1 := "t22", in2 := 2)
      { S7_Templates := "SrcType := Int" } EQ_Contact(in1 := "t33", in2 := 2)
   END_RUNG wire#w1
   RUNG wire#powerrail
      { S7_Templates := "SrcType := Int" } EQ_Contact(in1 := "t00", in2 := 2)
      { S7_Templates := "SrcType := Int" } EQ_Contact(in1 := "t10", in2 := 2)
      { S7_Templates := "SrcType := Int" } EQ_Contact(in1 := "t20", in2 := 2)
      { S7_Templates := "SrcType := Int" } EQ_Contact(in1 := "t30", in2 := 2)
   END_RUNG wire#w1
   RUNG wire#powerrail
      { S7_Templates := "SrcType := Int" } EQ_Contact(in1 := "t10", in2 := 2)
      { S7_Templates := "SrcType := Int" } EQ_Contact(in1 := "t11", in2 := 2)
      { S7_Templates := "SrcType := Int" } EQ_Contact(in1 := "t12", in2 := 2)
      { S7_Templates := "SrcType := Int" } EQ_Contact(in1 := "t13", in2 := 2)
   END_RUNG wire#w1
   RUNG wire#powerrail
      { S7_Templates := "SrcType := Int" } EQ_Contact(in1 := "t01", in2 := 2)
      { S7_Templates := "SrcType := Int" } EQ_Contact(in1 := "t11", in2 := 2)
      { S7_Templates := "SrcType := Int" } EQ_Contact(in1 := "t21", in2 := 2)
      { S7_Templates := "SrcType := Int" } EQ_Contact(in1 := "t31", in2 := 2)
   END_RUNG wire#w1
   RUNG wire#powerrail
      { S7_Templates := "SrcType := Int" } EQ_Contact(in1 := "t02", in2 := 2)
      { S7_Templates := "SrcType := Int" } EQ_Contact(in1 := "t12", in2 := 2)
      { S7_Templates := "SrcType := Int" } EQ_Contact(in1 := "t22", in2 := 2)
      { S7_Templates := "SrcType := Int" } EQ_Contact(in1 := "t32", in2 := 2)
   END_RUNG wire#w1
   RUNG wire#powerrail
      { S7_Templates := "SrcType := Int" } EQ_Contact(in1 := "t03", in2 := 2)
      { S7_Templates := "SrcType := Int" } EQ_Contact(in1 := "t12", in2 := 2)
      { S7_Templates := "SrcType := Int" } EQ_Contact(in1 := "t21", in2 := 2)
      { S7_Templates := "SrcType := Int" } EQ_Contact(in1 := "t30", in2 := 2)
   END_RUNG wire#w1
   RUNG wire#powerrail
      { S7_Templates := "SrcType := Int" } EQ_Contact(in1 := "t20", in2 := 2)
      { S7_Templates := "SrcType := Int" } EQ_Contact(in1 := "t21", in2 := 2)
      { S7_Templates := "SrcType := Int" } EQ_Contact(in1 := "t22", in2 := 2)
      { S7_Templates := "SrcType := Int" } EQ_Contact(in1 := "t23", in2 := 2)
   END_RUNG wire#w1
   RUNG wire#powerrail
      { S7_Templates := "SrcType := Int" } EQ_Contact(in1 := "t30", in2 := 2)
      { S7_Templates := "SrcType := Int" } EQ_Contact(in1 := "t31", in2 := 2)
      { S7_Templates := "SrcType := Int" } EQ_Contact(in1 := "t32", in2 := 2)
      { S7_Templates := "SrcType := Int" } EQ_Contact(in1 := "t33", in2 := 2)
   END_RUNG wire#w1
   RUNG wire#powerrail
      { S7_Templates := "SrcType := Int" } EQ_Contact(in1 := "t03", in2 := 2)
      { S7_Templates := "SrcType := Int" } EQ_Contact(in1 := "t13", in2 := 2)
      { S7_Templates := "SrcType := Int" } EQ_Contact(in1 := "t23", in2 := 2)
      { S7_Templates := "SrcType := Int" } EQ_Contact(in1 := "t33", in2 := 2)
   END_RUNG wire#w1
   RUNG wire#w1
      S_Coil( #Stop )
   END_RUNG
   // the same network as SCL:
   IF (("t00" = 2) AND ("t01" = 2) AND ("t02" = 2) AND ("t03" = 2)) OR (("t00" = 2) AND ("t11" = 2) AND ("t22" = 2) AND ("t33" = 2)) OR (("t00" = 2) AND ("t10" = 2) AND ("t20" = 2) AND ("t30" = 2)) OR (("t10" = 2) AND ("t11" = 2) AND ("t12" = 2) AND ("t13" = 2)) OR (("t01" = 2) AND ("t11" = 2) AND ("t21" = 2) AND ("t31" = 2)) OR (("t02" = 2) AND ("t12" = 2) AND ("t22" = 2) AND ("t32" = 2)) OR (("t03" = 2) AND ("t12" = 2) AND ("t21" = 2) AND ("t30" = 2)) OR (("t20" = 2) AND ("t21" = 2) AND ("t22" = 2) AND ("t23" = 2)) OR (("t30" = 2) AND ("t31" = 2) AND ("t32" = 2) AND ("t33" = 2)) OR (("t03" = 2) AND ("t13" = 2) AND ("t23" = 2) AND ("t33" = 2)) THEN
       #WinValue := 2;
       #Stop := TRUE;
   END_IF;
END_REGION
END_FUNCTION

// folder: 4x4/4x4PvC

FUNCTION "4x4PvCGame" : Void   // FC9, LAD
{ S7_Optimized_Access := 'TRUE' }
VERSION : 0.1
   VAR_TEMP
      temp00 : Bool;
      temp01 : Bool;
      temp02 : Bool;
      temp10 : Bool;
      temp11 : Bool;
      temp12 : Bool;
      temp20 : Bool;
      temp21 : Bool;
      temp22 : Bool;
      temp03 : Bool;
      temp13 : Bool;
      temp23 : Bool;
      temp33 : Bool;
      temp32 : Bool;
      temp31 : Bool;
      temp30 : Bool;
      WINX : Bool;
      WINO : Bool;
      rngValue : Int;
      tempplayer : Bool;
      tempBot : Bool;
      tempMove : Bool;
   END_VAR
   VAR_TEMP   // added for the SCL form of the ladder/FBD networks
      _w1 : Bool;
      _w2 : Bool;
      _w3 : Bool;
      _w4 : Bool;
      _w5 : Bool;
      _w6 : Bool;
      _w7 : Bool;
      _w8 : Bool;
      _w9 : Bool;
      _w10 : Bool;
      _w11 : Bool;
      _w12 : Bool;
      _w13 : Bool;
      _w14 : Bool;
      _w15 : Bool;
      _w16 : Bool;
      _w17 : Bool;
   END_VAR
BEGIN

REGION Network 1
   // Ruch gracza
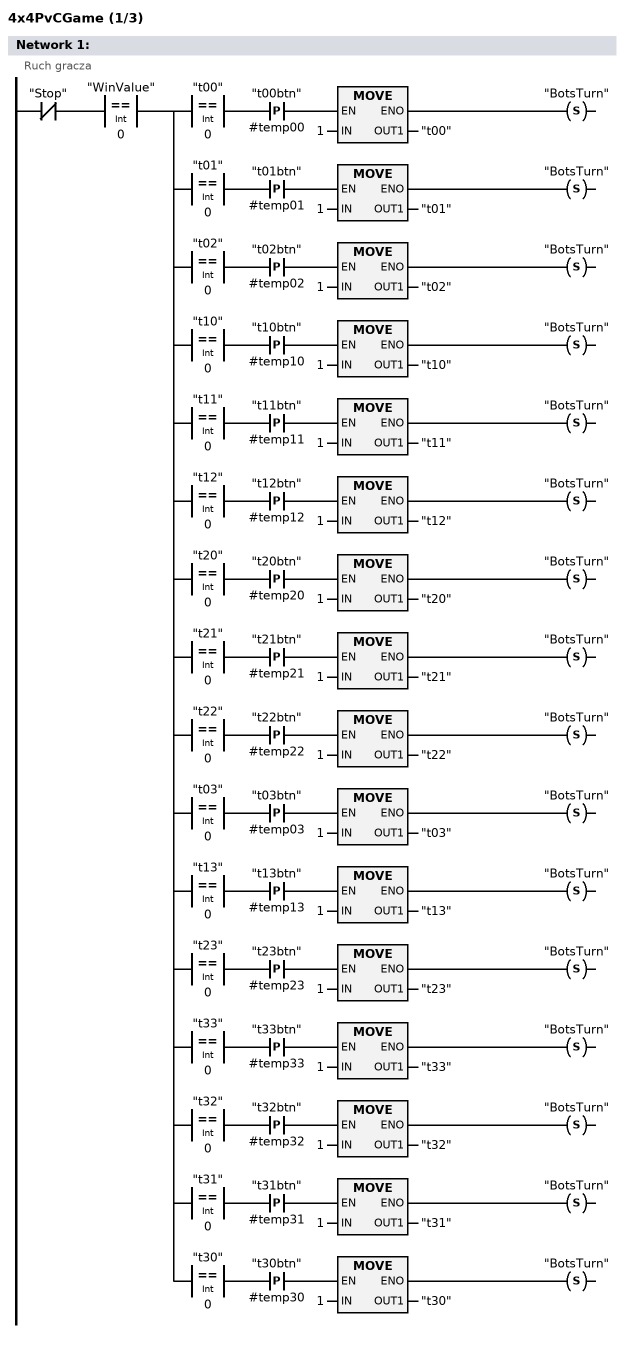
   RUNG wire#powerrail
      I_Contact( "Stop" )
      { S7_Templates := "SrcType := Int" } EQ_Contact(in1 := "WinValue", in2 := 0)
      wire#w1
      { S7_Templates := "SrcType := Int" } EQ_Contact(in1 := "t00", in2 := 0)
      P_Contact(operand := "t00btn", bit := #temp00)
      Move(in := 1, out1 => "t00")
      S_Coil( "BotsTurn" )
   END_RUNG
   RUNG wire#w1
      { S7_Templates := "SrcType := Int" } EQ_Contact(in1 := "t01", in2 := 0)
      P_Contact(operand := "t01btn", bit := #temp01)
      Move(in := 1, out1 => "t01")
      S_Coil( "BotsTurn" )
   END_RUNG
   RUNG wire#w1
      { S7_Templates := "SrcType := Int" } EQ_Contact(in1 := "t02", in2 := 0)
      P_Contact(operand := "t02btn", bit := #temp02)
      Move(in := 1, out1 => "t02")
      S_Coil( "BotsTurn" )
   END_RUNG
   RUNG wire#w1
      { S7_Templates := "SrcType := Int" } EQ_Contact(in1 := "t10", in2 := 0)
      P_Contact(operand := "t10btn", bit := #temp10)
      Move(in := 1, out1 => "t10")
      S_Coil( "BotsTurn" )
   END_RUNG
   RUNG wire#w1
      { S7_Templates := "SrcType := Int" } EQ_Contact(in1 := "t11", in2 := 0)
      P_Contact(operand := "t11btn", bit := #temp11)
      Move(in := 1, out1 => "t11")
      S_Coil( "BotsTurn" )
   END_RUNG
   RUNG wire#w1
      { S7_Templates := "SrcType := Int" } EQ_Contact(in1 := "t12", in2 := 0)
      P_Contact(operand := "t12btn", bit := #temp12)
      Move(in := 1, out1 => "t12")
      S_Coil( "BotsTurn" )
   END_RUNG
   RUNG wire#w1
      { S7_Templates := "SrcType := Int" } EQ_Contact(in1 := "t20", in2 := 0)
      P_Contact(operand := "t20btn", bit := #temp20)
      Move(in := 1, out1 => "t20")
      S_Coil( "BotsTurn" )
   END_RUNG
   RUNG wire#w1
      { S7_Templates := "SrcType := Int" } EQ_Contact(in1 := "t21", in2 := 0)
      P_Contact(operand := "t21btn", bit := #temp21)
      Move(in := 1, out1 => "t21")
      S_Coil( "BotsTurn" )
   END_RUNG
   RUNG wire#w1
      { S7_Templates := "SrcType := Int" } EQ_Contact(in1 := "t22", in2 := 0)
      P_Contact(operand := "t22btn", bit := #temp22)
      Move(in := 1, out1 => "t22")
      S_Coil( "BotsTurn" )
   END_RUNG
   RUNG wire#w1
      { S7_Templates := "SrcType := Int" } EQ_Contact(in1 := "t03", in2 := 0)
      P_Contact(operand := "t03btn", bit := #temp03)
      Move(in := 1, out1 => "t03")
      S_Coil( "BotsTurn" )
   END_RUNG
   RUNG wire#w1
      { S7_Templates := "SrcType := Int" } EQ_Contact(in1 := "t13", in2 := 0)
      P_Contact(operand := "t13btn", bit := #temp13)
      Move(in := 1, out1 => "t13")
      S_Coil( "BotsTurn" )
   END_RUNG
   RUNG wire#w1
      { S7_Templates := "SrcType := Int" } EQ_Contact(in1 := "t23", in2 := 0)
      P_Contact(operand := "t23btn", bit := #temp23)
      Move(in := 1, out1 => "t23")
      S_Coil( "BotsTurn" )
   END_RUNG
   RUNG wire#w1
      { S7_Templates := "SrcType := Int" } EQ_Contact(in1 := "t33", in2 := 0)
      P_Contact(operand := "t33btn", bit := #temp33)
      Move(in := 1, out1 => "t33")
      S_Coil( "BotsTurn" )
   END_RUNG
   RUNG wire#w1
      { S7_Templates := "SrcType := Int" } EQ_Contact(in1 := "t32", in2 := 0)
      P_Contact(operand := "t32btn", bit := #temp32)
      Move(in := 1, out1 => "t32")
      S_Coil( "BotsTurn" )
   END_RUNG
   RUNG wire#w1
      { S7_Templates := "SrcType := Int" } EQ_Contact(in1 := "t31", in2 := 0)
      P_Contact(operand := "t31btn", bit := #temp31)
      Move(in := 1, out1 => "t31")
      S_Coil( "BotsTurn" )
   END_RUNG
   RUNG wire#w1
      { S7_Templates := "SrcType := Int" } EQ_Contact(in1 := "t30", in2 := 0)
      P_Contact(operand := "t30btn", bit := #temp30)
      Move(in := 1, out1 => "t30")
      S_Coil( "BotsTurn" )
   END_RUNG
   // the same network as SCL:
   #_w1 := NOT "Stop" AND ("WinValue" = 0);
   #_w2 := #_w1 AND ("t00" = 0) AND "t00btn" AND NOT #temp00;   // rising edge of "t00btn"
   #temp00 := "t00btn";
   IF #_w2 THEN
       "t00" := 1;
       "BotsTurn" := TRUE;
   END_IF;
   #_w3 := #_w1 AND ("t01" = 0) AND "t01btn" AND NOT #temp01;   // rising edge of "t01btn"
   #temp01 := "t01btn";
   IF #_w3 THEN
       "t01" := 1;
       "BotsTurn" := TRUE;
   END_IF;
   #_w4 := #_w1 AND ("t02" = 0) AND "t02btn" AND NOT #temp02;   // rising edge of "t02btn"
   #temp02 := "t02btn";
   IF #_w4 THEN
       "t02" := 1;
       "BotsTurn" := TRUE;
   END_IF;
   #_w5 := #_w1 AND ("t10" = 0) AND "t10btn" AND NOT #temp10;   // rising edge of "t10btn"
   #temp10 := "t10btn";
   IF #_w5 THEN
       "t10" := 1;
       "BotsTurn" := TRUE;
   END_IF;
   #_w6 := #_w1 AND ("t11" = 0) AND "t11btn" AND NOT #temp11;   // rising edge of "t11btn"
   #temp11 := "t11btn";
   IF #_w6 THEN
       "t11" := 1;
       "BotsTurn" := TRUE;
   END_IF;
   #_w7 := #_w1 AND ("t12" = 0) AND "t12btn" AND NOT #temp12;   // rising edge of "t12btn"
   #temp12 := "t12btn";
   IF #_w7 THEN
       "t12" := 1;
       "BotsTurn" := TRUE;
   END_IF;
   #_w8 := #_w1 AND ("t20" = 0) AND "t20btn" AND NOT #temp20;   // rising edge of "t20btn"
   #temp20 := "t20btn";
   IF #_w8 THEN
       "t20" := 1;
       "BotsTurn" := TRUE;
   END_IF;
   #_w9 := #_w1 AND ("t21" = 0) AND "t21btn" AND NOT #temp21;   // rising edge of "t21btn"
   #temp21 := "t21btn";
   IF #_w9 THEN
       "t21" := 1;
       "BotsTurn" := TRUE;
   END_IF;
   #_w10 := #_w1 AND ("t22" = 0) AND "t22btn" AND NOT #temp22;   // rising edge of "t22btn"
   #temp22 := "t22btn";
   IF #_w10 THEN
       "t22" := 1;
       "BotsTurn" := TRUE;
   END_IF;
   #_w11 := #_w1 AND ("t03" = 0) AND "t03btn" AND NOT #temp03;   // rising edge of "t03btn"
   #temp03 := "t03btn";
   IF #_w11 THEN
       "t03" := 1;
       "BotsTurn" := TRUE;
   END_IF;
   #_w12 := #_w1 AND ("t13" = 0) AND "t13btn" AND NOT #temp13;   // rising edge of "t13btn"
   #temp13 := "t13btn";
   IF #_w12 THEN
       "t13" := 1;
       "BotsTurn" := TRUE;
   END_IF;
   #_w13 := #_w1 AND ("t23" = 0) AND "t23btn" AND NOT #temp23;   // rising edge of "t23btn"
   #temp23 := "t23btn";
   IF #_w13 THEN
       "t23" := 1;
       "BotsTurn" := TRUE;
   END_IF;
   #_w14 := #_w1 AND ("t33" = 0) AND "t33btn" AND NOT #temp33;   // rising edge of "t33btn"
   #temp33 := "t33btn";
   IF #_w14 THEN
       "t33" := 1;
       "BotsTurn" := TRUE;
   END_IF;
   #_w15 := #_w1 AND ("t32" = 0) AND "t32btn" AND NOT #temp32;   // rising edge of "t32btn"
   #temp32 := "t32btn";
   IF #_w15 THEN
       "t32" := 1;
       "BotsTurn" := TRUE;
   END_IF;
   #_w16 := #_w1 AND ("t31" = 0) AND "t31btn" AND NOT #temp31;   // rising edge of "t31btn"
   #temp31 := "t31btn";
   IF #_w16 THEN
       "t31" := 1;
       "BotsTurn" := TRUE;
   END_IF;
   #_w17 := #_w1 AND ("t30" = 0) AND "t30btn" AND NOT #temp30;   // rising edge of "t30btn"
   #temp30 := "t30btn";
   IF #_w17 THEN
       "t30" := 1;
       "BotsTurn" := TRUE;
   END_IF;
END_REGION

REGION Network 2
   // Ruch komputera
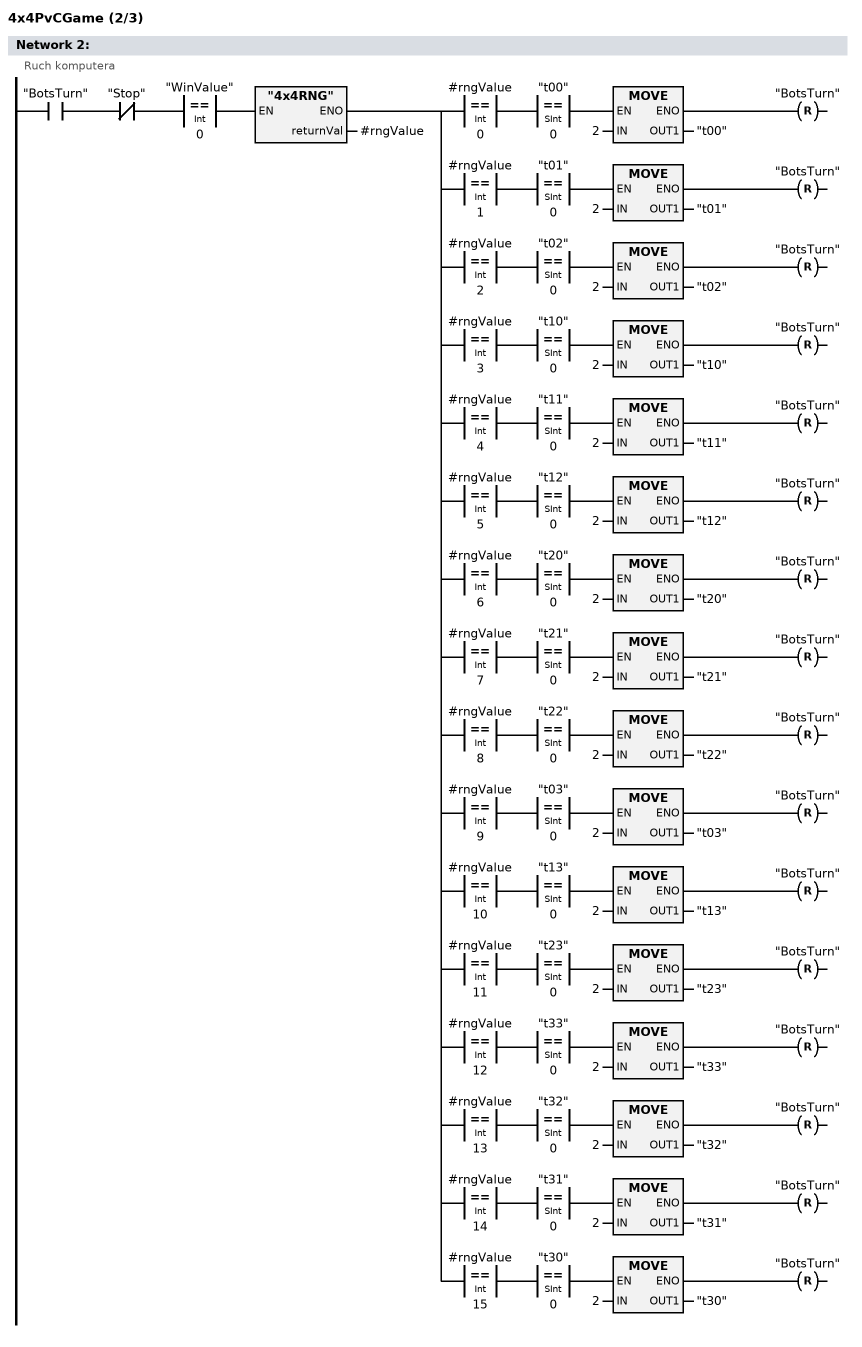
   RUNG wire#powerrail
      Contact( "BotsTurn" )
      I_Contact( "Stop" )
      { S7_Templates := "SrcType := Int" } EQ_Contact(in1 := "WinValue", in2 := 0)
      "4x4RNG"(returnVal => #rngValue)
      wire#w1
      { S7_Templates := "SrcType := Int" } EQ_Contact(in1 := #rngValue, in2 := 0)
      { S7_Templates := "SrcType := SInt" } EQ_Contact(in1 := "t00", in2 := 0)
      Move(in := 2, out1 => "t00")
      R_Coil( "BotsTurn" )
   END_RUNG
   RUNG wire#w1
      { S7_Templates := "SrcType := Int" } EQ_Contact(in1 := #rngValue, in2 := 1)
      { S7_Templates := "SrcType := SInt" } EQ_Contact(in1 := "t01", in2 := 0)
      Move(in := 2, out1 => "t01")
      R_Coil( "BotsTurn" )
   END_RUNG
   RUNG wire#w1
      { S7_Templates := "SrcType := Int" } EQ_Contact(in1 := #rngValue, in2 := 2)
      { S7_Templates := "SrcType := SInt" } EQ_Contact(in1 := "t02", in2 := 0)
      Move(in := 2, out1 => "t02")
      R_Coil( "BotsTurn" )
   END_RUNG
   RUNG wire#w1
      { S7_Templates := "SrcType := Int" } EQ_Contact(in1 := #rngValue, in2 := 3)
      { S7_Templates := "SrcType := SInt" } EQ_Contact(in1 := "t10", in2 := 0)
      Move(in := 2, out1 => "t10")
      R_Coil( "BotsTurn" )
   END_RUNG
   RUNG wire#w1
      { S7_Templates := "SrcType := Int" } EQ_Contact(in1 := #rngValue, in2 := 4)
      { S7_Templates := "SrcType := SInt" } EQ_Contact(in1 := "t11", in2 := 0)
      Move(in := 2, out1 => "t11")
      R_Coil( "BotsTurn" )
   END_RUNG
   RUNG wire#w1
      { S7_Templates := "SrcType := Int" } EQ_Contact(in1 := #rngValue, in2 := 5)
      { S7_Templates := "SrcType := SInt" } EQ_Contact(in1 := "t12", in2 := 0)
      Move(in := 2, out1 => "t12")
      R_Coil( "BotsTurn" )
   END_RUNG
   RUNG wire#w1
      { S7_Templates := "SrcType := Int" } EQ_Contact(in1 := #rngValue, in2 := 6)
      { S7_Templates := "SrcType := SInt" } EQ_Contact(in1 := "t20", in2 := 0)
      Move(in := 2, out1 => "t20")
      R_Coil( "BotsTurn" )
   END_RUNG
   RUNG wire#w1
      { S7_Templates := "SrcType := Int" } EQ_Contact(in1 := #rngValue, in2 := 7)
      { S7_Templates := "SrcType := SInt" } EQ_Contact(in1 := "t21", in2 := 0)
      Move(in := 2, out1 => "t21")
      R_Coil( "BotsTurn" )
   END_RUNG
   RUNG wire#w1
      { S7_Templates := "SrcType := Int" } EQ_Contact(in1 := #rngValue, in2 := 8)
      { S7_Templates := "SrcType := SInt" } EQ_Contact(in1 := "t22", in2 := 0)
      Move(in := 2, out1 => "t22")
      R_Coil( "BotsTurn" )
   END_RUNG
   RUNG wire#w1
      { S7_Templates := "SrcType := Int" } EQ_Contact(in1 := #rngValue, in2 := 9)
      { S7_Templates := "SrcType := SInt" } EQ_Contact(in1 := "t03", in2 := 0)
      Move(in := 2, out1 => "t03")
      R_Coil( "BotsTurn" )
   END_RUNG
   RUNG wire#w1
      { S7_Templates := "SrcType := Int" } EQ_Contact(in1 := #rngValue, in2 := 10)
      { S7_Templates := "SrcType := SInt" } EQ_Contact(in1 := "t13", in2 := 0)
      Move(in := 2, out1 => "t13")
      R_Coil( "BotsTurn" )
   END_RUNG
   RUNG wire#w1
      { S7_Templates := "SrcType := Int" } EQ_Contact(in1 := #rngValue, in2 := 11)
      { S7_Templates := "SrcType := SInt" } EQ_Contact(in1 := "t23", in2 := 0)
      Move(in := 2, out1 => "t23")
      R_Coil( "BotsTurn" )
   END_RUNG
   RUNG wire#w1
      { S7_Templates := "SrcType := Int" } EQ_Contact(in1 := #rngValue, in2 := 12)
      { S7_Templates := "SrcType := SInt" } EQ_Contact(in1 := "t33", in2 := 0)
      Move(in := 2, out1 => "t33")
      R_Coil( "BotsTurn" )
   END_RUNG
   RUNG wire#w1
      { S7_Templates := "SrcType := Int" } EQ_Contact(in1 := #rngValue, in2 := 13)
      { S7_Templates := "SrcType := SInt" } EQ_Contact(in1 := "t32", in2 := 0)
      Move(in := 2, out1 => "t32")
      R_Coil( "BotsTurn" )
   END_RUNG
   RUNG wire#w1
      { S7_Templates := "SrcType := Int" } EQ_Contact(in1 := #rngValue, in2 := 14)
      { S7_Templates := "SrcType := SInt" } EQ_Contact(in1 := "t31", in2 := 0)
      Move(in := 2, out1 => "t31")
      R_Coil( "BotsTurn" )
   END_RUNG
   RUNG wire#w1
      { S7_Templates := "SrcType := Int" } EQ_Contact(in1 := #rngValue, in2 := 15)
      { S7_Templates := "SrcType := SInt" } EQ_Contact(in1 := "t30", in2 := 0)
      Move(in := 2, out1 => "t30")
      R_Coil( "BotsTurn" )
   END_RUNG
   // the same network as SCL:
   "4x4RNG"(EN := "BotsTurn" AND NOT "Stop" AND ("WinValue" = 0), returnVal => #rngValue, ENO => #_w1);
   #_w2 := #_w1 AND (#rngValue = 0) AND ("t00" = 0);
   IF #_w2 THEN
       "t00" := 2;
       "BotsTurn" := FALSE;
   END_IF;
   #_w3 := #_w1 AND (#rngValue = 1) AND ("t01" = 0);
   IF #_w3 THEN
       "t01" := 2;
       "BotsTurn" := FALSE;
   END_IF;
   #_w4 := #_w1 AND (#rngValue = 2) AND ("t02" = 0);
   IF #_w4 THEN
       "t02" := 2;
       "BotsTurn" := FALSE;
   END_IF;
   #_w5 := #_w1 AND (#rngValue = 3) AND ("t10" = 0);
   IF #_w5 THEN
       "t10" := 2;
       "BotsTurn" := FALSE;
   END_IF;
   #_w6 := #_w1 AND (#rngValue = 4) AND ("t11" = 0);
   IF #_w6 THEN
       "t11" := 2;
       "BotsTurn" := FALSE;
   END_IF;
   #_w7 := #_w1 AND (#rngValue = 5) AND ("t12" = 0);
   IF #_w7 THEN
       "t12" := 2;
       "BotsTurn" := FALSE;
   END_IF;
   #_w8 := #_w1 AND (#rngValue = 6) AND ("t20" = 0);
   IF #_w8 THEN
       "t20" := 2;
       "BotsTurn" := FALSE;
   END_IF;
   #_w9 := #_w1 AND (#rngValue = 7) AND ("t21" = 0);
   IF #_w9 THEN
       "t21" := 2;
       "BotsTurn" := FALSE;
   END_IF;
   #_w10 := #_w1 AND (#rngValue = 8) AND ("t22" = 0);
   IF #_w10 THEN
       "t22" := 2;
       "BotsTurn" := FALSE;
   END_IF;
   #_w11 := #_w1 AND (#rngValue = 9) AND ("t03" = 0);
   IF #_w11 THEN
       "t03" := 2;
       "BotsTurn" := FALSE;
   END_IF;
   #_w12 := #_w1 AND (#rngValue = 10) AND ("t13" = 0);
   IF #_w12 THEN
       "t13" := 2;
       "BotsTurn" := FALSE;
   END_IF;
   #_w13 := #_w1 AND (#rngValue = 11) AND ("t23" = 0);
   IF #_w13 THEN
       "t23" := 2;
       "BotsTurn" := FALSE;
   END_IF;
   #_w14 := #_w1 AND (#rngValue = 12) AND ("t33" = 0);
   IF #_w14 THEN
       "t33" := 2;
       "BotsTurn" := FALSE;
   END_IF;
   #_w15 := #_w1 AND (#rngValue = 13) AND ("t32" = 0);
   IF #_w15 THEN
       "t32" := 2;
       "BotsTurn" := FALSE;
   END_IF;
   #_w16 := #_w1 AND (#rngValue = 14) AND ("t31" = 0);
   IF #_w16 THEN
       "t31" := 2;
       "BotsTurn" := FALSE;
   END_IF;
   #_w17 := #_w1 AND (#rngValue = 15) AND ("t30" = 0);
   IF #_w17 THEN
       "t30" := 2;
       "BotsTurn" := FALSE;
   END_IF;
END_REGION

REGION Network 3
   // Sprawdzanie wygranej
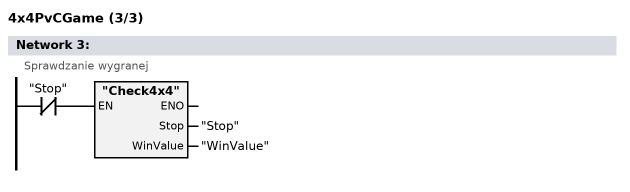
   RUNG wire#powerrail
      I_Contact( "Stop" )
      "Check4x4"(Stop => "Stop", WinValue => "WinValue")
   END_RUNG
   // the same network as SCL:
   IF NOT "Stop" THEN "Check4x4"(Stop => "Stop", WinValue => "WinValue"); END_IF;
END_REGION
END_FUNCTION

FUNCTION "4x4RNG" : Void   // FC10, LAD
{ S7_Optimized_Access := 'TRUE' }
VERSION : 0.1
   VAR_OUTPUT
      returnVal : Int;
   END_VAR
   VAR_TEMP
      val : Int;
      reset : Bool;
      Stop : Bool;
      datetemp : DTL;
   END_VAR
BEGIN

REGION Network 1
   // Generowanie losowego pola
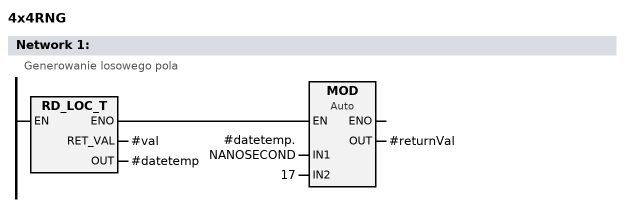
   // ENO of a box is taken as its EN; it also drops when the box reports an error
   #val := RD_LOC_T(OUT => #datetemp);
   #returnVal := #datetemp.NANOSECOND MOD 17;
END_REGION
END_FUNCTION

// folder: 4x4/4x4PvP

FUNCTION "4x4PvPGame" : Void   // FC7, LAD
{ S7_Optimized_Access := 'TRUE' }
VERSION : 0.1
   VAR_TEMP
      temp00 : Bool;
      temp01 : Bool;
      temp02 : Bool;
      temp10 : Bool;
      temp11 : Bool;
      temp12 : Bool;
      temp20 : Bool;
      temp21 : Bool;
      temp22 : Bool;
      temp03 : Bool;
      temp13 : Bool;
      temp23 : Bool;
      temp33 : Bool;
      temp32 : Bool;
      temp31 : Bool;
      temp30 : Bool;
      WINX : Bool;
      WINO : Bool;
   END_VAR
   VAR_TEMP   // added for the SCL form of the ladder/FBD networks
      _w1 : Bool;
      _w2 : Bool;
      _w3 : Bool;
      _w4 : Bool;
      _w5 : Bool;
      _w6 : Bool;
      _w7 : Bool;
      _w8 : Bool;
      _w9 : Bool;
      _w10 : Bool;
      _w11 : Bool;
      _w12 : Bool;
      _w13 : Bool;
      _w14 : Bool;
      _w15 : Bool;
      _w16 : Bool;
      _w17 : Bool;
   END_VAR
BEGIN

REGION Network 1
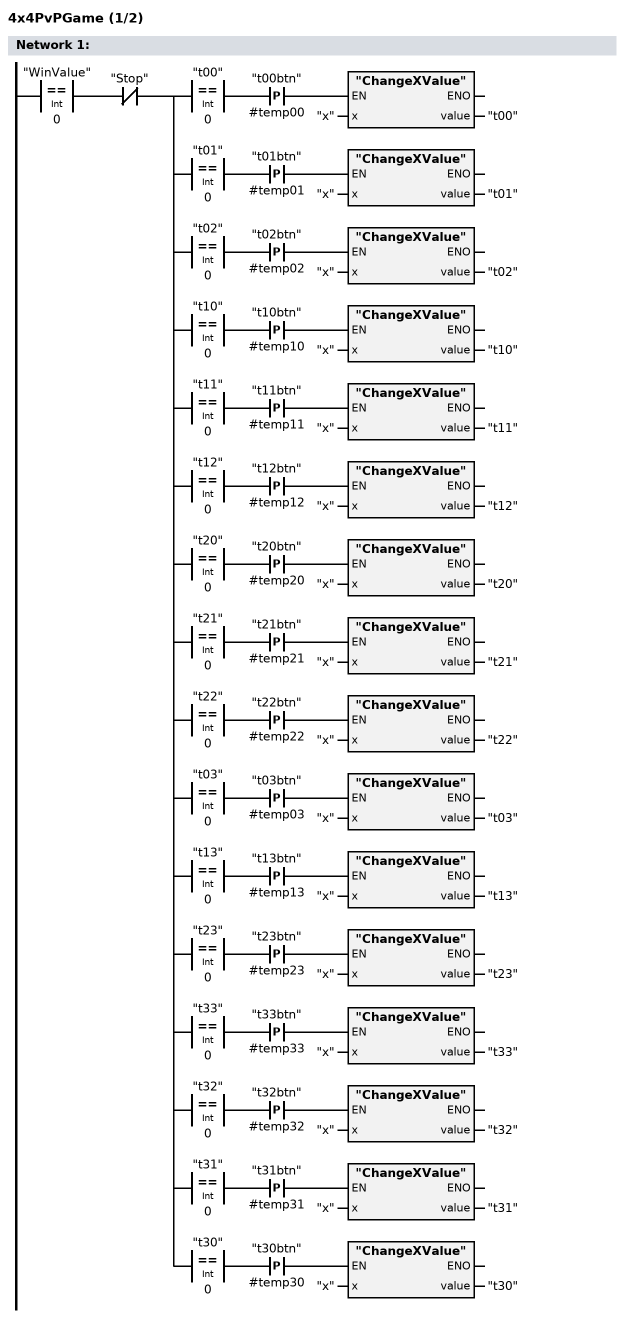
   RUNG wire#powerrail
      { S7_Templates := "SrcType := Int" } EQ_Contact(in1 := "WinValue", in2 := 0)
      I_Contact( "Stop" )
      wire#w1
      { S7_Templates := "SrcType := Int" } EQ_Contact(in1 := "t00", in2 := 0)
      P_Contact(operand := "t00btn", bit := #temp00)
      "ChangeXValue"(x := "x", value => "t00")
   END_RUNG
   RUNG wire#w1
      { S7_Templates := "SrcType := Int" } EQ_Contact(in1 := "t01", in2 := 0)
      P_Contact(operand := "t01btn", bit := #temp01)
      "ChangeXValue"(x := "x", value => "t01")
   END_RUNG
   RUNG wire#w1
      { S7_Templates := "SrcType := Int" } EQ_Contact(in1 := "t02", in2 := 0)
      P_Contact(operand := "t02btn", bit := #temp02)
      "ChangeXValue"(x := "x", value => "t02")
   END_RUNG
   RUNG wire#w1
      { S7_Templates := "SrcType := Int" } EQ_Contact(in1 := "t10", in2 := 0)
      P_Contact(operand := "t10btn", bit := #temp10)
      "ChangeXValue"(x := "x", value => "t10")
   END_RUNG
   RUNG wire#w1
      { S7_Templates := "SrcType := Int" } EQ_Contact(in1 := "t11", in2 := 0)
      P_Contact(operand := "t11btn", bit := #temp11)
      "ChangeXValue"(x := "x", value => "t11")
   END_RUNG
   RUNG wire#w1
      { S7_Templates := "SrcType := Int" } EQ_Contact(in1 := "t12", in2 := 0)
      P_Contact(operand := "t12btn", bit := #temp12)
      "ChangeXValue"(x := "x", value => "t12")
   END_RUNG
   RUNG wire#w1
      { S7_Templates := "SrcType := Int" } EQ_Contact(in1 := "t20", in2 := 0)
      P_Contact(operand := "t20btn", bit := #temp20)
      "ChangeXValue"(x := "x", value => "t20")
   END_RUNG
   RUNG wire#w1
      { S7_Templates := "SrcType := Int" } EQ_Contact(in1 := "t21", in2 := 0)
      P_Contact(operand := "t21btn", bit := #temp21)
      "ChangeXValue"(x := "x", value => "t21")
   END_RUNG
   RUNG wire#w1
      { S7_Templates := "SrcType := Int" } EQ_Contact(in1 := "t22", in2 := 0)
      P_Contact(operand := "t22btn", bit := #temp22)
      "ChangeXValue"(x := "x", value => "t22")
   END_RUNG
   RUNG wire#w1
      { S7_Templates := "SrcType := Int" } EQ_Contact(in1 := "t03", in2 := 0)
      P_Contact(operand := "t03btn", bit := #temp03)
      "ChangeXValue"(x := "x", value => "t03")
   END_RUNG
   RUNG wire#w1
      { S7_Templates := "SrcType := Int" } EQ_Contact(in1 := "t13", in2 := 0)
      P_Contact(operand := "t13btn", bit := #temp13)
      "ChangeXValue"(x := "x", value => "t13")
   END_RUNG
   RUNG wire#w1
      { S7_Templates := "SrcType := Int" } EQ_Contact(in1 := "t23", in2 := 0)
      P_Contact(operand := "t23btn", bit := #temp23)
      "ChangeXValue"(x := "x", value => "t23")
   END_RUNG
   RUNG wire#w1
      { S7_Templates := "SrcType := Int" } EQ_Contact(in1 := "t33", in2 := 0)
      P_Contact(operand := "t33btn", bit := #temp33)
      "ChangeXValue"(x := "x", value => "t33")
   END_RUNG
   RUNG wire#w1
      { S7_Templates := "SrcType := Int" } EQ_Contact(in1 := "t32", in2 := 0)
      P_Contact(operand := "t32btn", bit := #temp32)
      "ChangeXValue"(x := "x", value => "t32")
   END_RUNG
   RUNG wire#w1
      { S7_Templates := "SrcType := Int" } EQ_Contact(in1 := "t31", in2 := 0)
      P_Contact(operand := "t31btn", bit := #temp31)
      "ChangeXValue"(x := "x", value => "t31")
   END_RUNG
   RUNG wire#w1
      { S7_Templates := "SrcType := Int" } EQ_Contact(in1 := "t30", in2 := 0)
      P_Contact(operand := "t30btn", bit := #temp30)
      "ChangeXValue"(x := "x", value => "t30")
   END_RUNG
   // the same network as SCL:
   #_w1 := ("WinValue" = 0) AND NOT "Stop";
   #_w2 := #_w1 AND ("t00" = 0) AND "t00btn" AND NOT #temp00;   // rising edge of "t00btn"
   #temp00 := "t00btn";
   IF #_w2 THEN "ChangeXValue"(x := "x", value => "t00"); END_IF;
   #_w3 := #_w1 AND ("t01" = 0) AND "t01btn" AND NOT #temp01;   // rising edge of "t01btn"
   #temp01 := "t01btn";
   IF #_w3 THEN "ChangeXValue"(x := "x", value => "t01"); END_IF;
   #_w4 := #_w1 AND ("t02" = 0) AND "t02btn" AND NOT #temp02;   // rising edge of "t02btn"
   #temp02 := "t02btn";
   IF #_w4 THEN "ChangeXValue"(x := "x", value => "t02"); END_IF;
   #_w5 := #_w1 AND ("t10" = 0) AND "t10btn" AND NOT #temp10;   // rising edge of "t10btn"
   #temp10 := "t10btn";
   IF #_w5 THEN "ChangeXValue"(x := "x", value => "t10"); END_IF;
   #_w6 := #_w1 AND ("t11" = 0) AND "t11btn" AND NOT #temp11;   // rising edge of "t11btn"
   #temp11 := "t11btn";
   IF #_w6 THEN "ChangeXValue"(x := "x", value => "t11"); END_IF;
   #_w7 := #_w1 AND ("t12" = 0) AND "t12btn" AND NOT #temp12;   // rising edge of "t12btn"
   #temp12 := "t12btn";
   IF #_w7 THEN "ChangeXValue"(x := "x", value => "t12"); END_IF;
   #_w8 := #_w1 AND ("t20" = 0) AND "t20btn" AND NOT #temp20;   // rising edge of "t20btn"
   #temp20 := "t20btn";
   IF #_w8 THEN "ChangeXValue"(x := "x", value => "t20"); END_IF;
   #_w9 := #_w1 AND ("t21" = 0) AND "t21btn" AND NOT #temp21;   // rising edge of "t21btn"
   #temp21 := "t21btn";
   IF #_w9 THEN "ChangeXValue"(x := "x", value => "t21"); END_IF;
   #_w10 := #_w1 AND ("t22" = 0) AND "t22btn" AND NOT #temp22;   // rising edge of "t22btn"
   #temp22 := "t22btn";
   IF #_w10 THEN "ChangeXValue"(x := "x", value => "t22"); END_IF;
   #_w11 := #_w1 AND ("t03" = 0) AND "t03btn" AND NOT #temp03;   // rising edge of "t03btn"
   #temp03 := "t03btn";
   IF #_w11 THEN "ChangeXValue"(x := "x", value => "t03"); END_IF;
   #_w12 := #_w1 AND ("t13" = 0) AND "t13btn" AND NOT #temp13;   // rising edge of "t13btn"
   #temp13 := "t13btn";
   IF #_w12 THEN "ChangeXValue"(x := "x", value => "t13"); END_IF;
   #_w13 := #_w1 AND ("t23" = 0) AND "t23btn" AND NOT #temp23;   // rising edge of "t23btn"
   #temp23 := "t23btn";
   IF #_w13 THEN "ChangeXValue"(x := "x", value => "t23"); END_IF;
   #_w14 := #_w1 AND ("t33" = 0) AND "t33btn" AND NOT #temp33;   // rising edge of "t33btn"
   #temp33 := "t33btn";
   IF #_w14 THEN "ChangeXValue"(x := "x", value => "t33"); END_IF;
   #_w15 := #_w1 AND ("t32" = 0) AND "t32btn" AND NOT #temp32;   // rising edge of "t32btn"
   #temp32 := "t32btn";
   IF #_w15 THEN "ChangeXValue"(x := "x", value => "t32"); END_IF;
   #_w16 := #_w1 AND ("t31" = 0) AND "t31btn" AND NOT #temp31;   // rising edge of "t31btn"
   #temp31 := "t31btn";
   IF #_w16 THEN "ChangeXValue"(x := "x", value => "t31"); END_IF;
   #_w17 := #_w1 AND ("t30" = 0) AND "t30btn" AND NOT #temp30;   // rising edge of "t30btn"
   #temp30 := "t30btn";
   IF #_w17 THEN "ChangeXValue"(x := "x", value => "t30"); END_IF;
END_REGION

REGION Network 2
   // Sprawdzanie wygranej
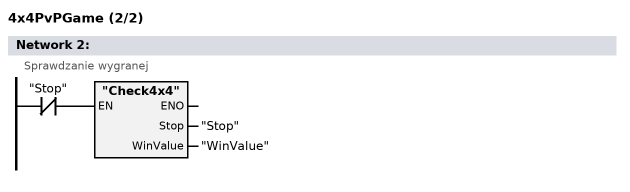
   RUNG wire#powerrail
      I_Contact( "Stop" )
      "Check4x4"(Stop => "Stop", WinValue => "WinValue")
   END_RUNG
   // the same network as SCL:
   IF NOT "Stop" THEN "Check4x4"(Stop => "Stop", WinValue => "WinValue"); END_IF;
END_REGION
END_FUNCTION

(* ===== HMI "HMI_RT_1" =====
system functions are stored by id; their names below are inferred from use
connection "HMI_Connection_1": ETHERNET, SMART_S7_1200_OMS

HMI tags "Default tag table"
   "Tag_ScreenNumber" : UInt, internal
   "x" : Bool = PLC x AT %M15.2, 500 ms
   "Reset" : Bool = PLC Reset AT %M12.1, 500 ms
   "WinValue" : SInt = PLC WinValue AT %MB36, 500 ms
   "GameType" : SInt = PLC GameType AT %MB17, 500 ms
   "BotsTurn" : Bool = PLC BotsTurn AT %M37.1, 1 s

HMI tags "3x3HmiTags"
   "t00_HMI" : SInt = PLC t00 AT %MB1, 100 ms
   "t01_HMI" : SInt = PLC t01 AT %MB2, 100 ms
   "t02_HMI" : SInt = PLC t02 AT %MB3, 100 ms
   "t10_HMI" : SInt = PLC t10 AT %MB4, 100 ms
   "t11_HMI" : SInt = PLC t11 AT %MB10, 100 ms
   "t12_HMI" : SInt = PLC t12 AT %MB13, 100 ms
   "t20_HMI" : SInt = PLC t20 AT %MB7, 100 ms
   "t21_HMI" : SInt = PLC t21 AT %MB8, 100 ms
   "t22_HMI" : SInt = PLC t22 AT %MB9, 100 ms
   "t00btn_HMI" : Bool = PLC t00btn AT %M5.1, 100 ms
   "t01btn_HMI" : Bool = PLC t01btn AT %M5.2, 100 ms
   "t02btn_HMI" : Bool = PLC t02btn AT %M5.3, 100 ms
   "t10btn_HMI" : Bool = PLC t10btn AT %M5.4, 100 ms
   "t11btn_HMI" : Bool = PLC t11btn AT %M5.5, 100 ms
   "t12btn_HMI" : Bool = PLC t12btn AT %M5.6, 100 ms
   "t20btn_HMI" : Bool = PLC t20btn AT %M5.7, 100 ms
   "t21btn_HMI" : Bool = PLC t21btn AT %M6.0, 100 ms
   "t22btn_HMI" : Bool = PLC t22btn AT %M6.1, 100 ms
   "t03_HMI" : SInt = PLC t03 AT %MB46, 100 ms
   "t13_HMI" : SInt = PLC t13 AT %MB38, 100 ms
   "t23_HMI" : SInt = PLC t23 AT %MB39, 100 ms
   "t33_HMI" : SInt = PLC t33 AT %MB40, 100 ms
   "t32_HMI" : SInt = PLC t32 AT %MB41, 100 ms
   "t31_HMI" : SInt = PLC t31 AT %MB42, 100 ms
   "t30_HMI" : SInt = PLC t30 AT %MB43, 100 ms
   "t03btn_HMI" : Bool = PLC t03btn AT %M44.0, 100 ms
   "t13btn_HMI" : Bool = PLC t13btn AT %M44.1, 100 ms
   "t23btn_HMI" : Bool = PLC t23btn AT %M44.2, 100 ms
   "t33btn_HMI" : Bool = PLC t33btn AT %M44.3, 100 ms
   "t32btn_HMI" : Bool = PLC t32btn AT %M44.4, 100 ms
   "t31btn_HMI" : Bool = PLC t31btn AT %M44.5, 100 ms
   "t30btn_HMI" : Bool = PLC t30btn AT %M44.6, 100 ms

text list "3x3_TextList": 0 ''; 1 'X'; 2 'O'

text list "WinInfo_TextList": 0 ''; 1 'Wygrał X! / X won! / X gewonnen!'; 2 'Wygrało O! / O won! / O gewonnen!'; 3 'Remis! / Draw! / Gleichstand'

Template "Menu" 320x240
   Button "Exit" at 266,202 size 52x37; TextOff 'Exit'; PictureOff "ExitRuntime_KTP600_Basic_color_PN"; PictureOn "ExitRuntime_KTP600_Basic_color_PN"
      on Release: StopRuntime(0)
   Button "Template_Button_3" at 54,202 size 212x37; TextOff 'Change the language / Zmiana języka / Ändere die Sprache'; TextList "3x3_TextList"
      on Click: function_fb9197e8(-1)
   Button "Start screen" at 1,202 size 52x37; TextOff 'Start screen'; PictureOff "NavigateHome_KTP600_Basic_color_PN"; PictureOn "NavigateHome_KTP600_Basic_color_PN"
      on Release: ActivateScreen("Root screen", 0); SetTag("GameType", 0)

screen "Root screen" 320x240, template "Menu"
   on GenerateScreen: SetTag("Tag_ScreenNumber", 1); SetTag("GameType", 0); SetBit("Reset")
   on ClearScreen: ResetBit("Reset")
   Button "Button_1" at 20,90 size 55x90; TextOff 'Gracz vs Gracz Player vs Player Spieler vs Spieler'
      on Release: SetTag("GameType", 1); ActivateScreen("3x3PvP", 0)
   Button "Button_2" at 84,90 size 55x90; TextOff 'Gracz vs Komputer Player vs Computer Spieler vs Computer'
      on Release: SetTag("GameType", 2); ActivateScreen("3x3PvC", 1)
   Button "Button_3" at 180,90 size 55x90; TextOff 'Gracz vs Gracz Player vs Player Spieler vs Spieler'
      on Release: SetTag("GameType", 3); ActivateScreen("4x4PvP", 1)
   Button "Button_4" at 243,90 size 55x90; TextOff 'Gracz vs Komputer Player vs Computer Spieler vs Computer'
      on Release: SetTag("GameType", 4); ActivateScreen("4x4PvC", 1)
   TextField "Text field_1" at 11,0 size 299x49; Text 'KÓŁKO I KRZYŻYK / TIC TAC TOE / DODELSCHACH'
   TextField "Text field_2" at 25,58 size 112x24; Text '3x3'
   TextField "Text field_3" at 185,58 size 112x24; Text '4x4'

screen "3x3PvP" 320x240, template "3x3Template"
   Button "Button_2" at 220,89 size 85x85; TextOff 'Reset'
      on Press: SetBit("Reset")
      on Release: ResetBit("Reset")
   Button "Button_3" at 15,15 size 50x50; TextOff 't00'; TextList "3x3_TextList"
      on Release: ResetBit("t00btn_HMI"); InvertBit("x")
      on Press: SetBit("t00btn_HMI")
      ProcessValue <- "t00(1)"
   Button "Button_5" at 135,15 size 50x50; TextOff 't02'; TextList "3x3_TextList"
      on Release: ResetBit("t02btn_HMI"); InvertBit("x")
      on Press: SetBit("t02btn_HMI")
      ProcessValue <- "t00(1)"
   Button "Button_1" at 75,15 size 50x50; TextOff 't01'; TextList "3x3_TextList"
      on Release: ResetBit("t01btn_HMI"); InvertBit("x")
      on Press: SetBit("t01btn_HMI")
      ProcessValue <- "t00(1)"
   Button "Button_6" at 15,75 size 50x50; TextOff 't10'; TextList "3x3_TextList"
      on Release: ResetBit("t10btn_HMI"); InvertBit("x")
      on Press: SetBit("t10btn_HMI")
      ProcessValue <- "t00(1)"
   Button "Button_7" at 135,75 size 50x50; TextOff 't12'; TextList "3x3_TextList"
      on Release: ResetBit("t12btn_HMI"); InvertBit("x")
      on Press: SetBit("t12btn_HMI")
      ProcessValue <- "t00(1)"
   Button "Button_8" at 75,75 size 50x50; TextOff 't11'; TextList "3x3_TextList"
      on Release: ResetBit("t11btn_HMI"); InvertBit("x")
      on Press: SetBit("t11btn_HMI")
      ProcessValue <- "t00(1)"
   Button "Button_9" at 15,135 size 50x50; TextOff 't20'; TextList "3x3_TextList"
      on Release: ResetBit("t20btn_HMI"); InvertBit("x")
      on Press: SetBit("t20btn_HMI")
      ProcessValue <- "t00(1)"
   Button "Button_10" at 135,135 size 50x50; TextOff 't22'; TextList "3x3_TextList"
      on Release: ResetBit("t22btn_HMI"); InvertBit("x")
      on Press: SetBit("t22btn_HMI")
      ProcessValue <- "t00(1)"
   Button "Button_11" at 75,135 size 50x50; TextOff 't21'; TextList "3x3_TextList"
      on Release: ResetBit("t21btn_HMI"); InvertBit("x")
      on Press: SetBit("t21btn_HMI")
      ProcessValue <- "t00(1)"
   SymbolicIOField "Symbolic I/O field_1" at 220,31 size 85x44; TextOff '0'; TextOn '1'; TextList "WinInfo_TextList"
      ProcessValue <- "WinValue"

screen "3x3PvC" 320x240, template "3x3Template"
   Button "Button_2" at 220,89 size 85x85; TextOff 'Reset'
      on Release: ResetBit("Reset")
      on Press: SetBit("Reset")
   Button "Button_3" at 15,15 size 50x50; TextOff 't00'; TextList "3x3_TextList"
      on Release: ResetBit("t00btn_HMI")
      on Press: SetBit("t00btn_HMI")
      ProcessValue <- "t00(1)"
   Button "Button_5" at 135,15 size 50x50; TextOff 't02'; TextList "3x3_TextList"
      on Release: ResetBit("t02btn_HMI")
      on Press: SetBit("t02btn_HMI")
      ProcessValue <- "t00(1)"
   Button "Button_1" at 75,15 size 50x50; TextOff 't01'; TextList "3x3_TextList"
      on Release: ResetBit("t01btn_HMI")
      on Press: SetBit("t01btn_HMI")
      ProcessValue <- "t00(1)"
   Button "Button_6" at 15,75 size 50x50; TextOff 't10'; TextList "3x3_TextList"
      on Release: ResetBit("t10btn_HMI")
      on Press: SetBit("t10btn_HMI")
      ProcessValue <- "t00(1)"
   Button "Button_7" at 135,75 size 50x50; TextOff 't12'; TextList "3x3_TextList"
      on Release: ResetBit("t12btn_HMI")
      on Press: SetBit("t12btn_HMI")
      ProcessValue <- "t00(1)"
   Button "Button_8" at 75,75 size 50x50; TextOff 't11'; TextList "3x3_TextList"
      on Release: ResetBit("t11btn_HMI")
      on Press: SetBit("t11btn_HMI")
      ProcessValue <- "t00(1)"
   Button "Button_9" at 15,135 size 50x50; TextOff 't20'; TextList "3x3_TextList"
      on Release: ResetBit("t20btn_HMI")
      on Press: SetBit("t20btn_HMI")
      ProcessValue <- "t00(1)"
   Button "Button_10" at 135,135 size 50x50; TextOff 't22'; TextList "3x3_TextList"
      on Release: ResetBit("t22btn_HMI")
      on Press: SetBit("t22btn_HMI")
      ProcessValue <- "t00(1)"
   Button "Button_11" at 75,135 size 50x50; TextOff 't21'; TextList "3x3_TextList"
      on Release: ResetBit("t21btn_HMI")
      on Press: SetBit("t21btn_HMI")
      ProcessValue <- "t00(1)"
   SymbolicIOField "Symbolic I/O field_1" at 220,31 size 85x44; TextOn '1'; TextOff '0'; TextList "WinInfo_TextList"
      ProcessValue <- "WinValue"

Template "3x3Template" 320x240
   Button "Exit" at 266,202 size 52x37; TextOn 'Exit'; TextOff 'Exit'; PictureOn "ExitRuntime_KTP600_Basic_color_PN"; PictureOff "ExitRuntime_KTP600_Basic_color_PN"
      on Release: StopRuntime(0)
   Button "Template_Button_3" at 54,202 size 212x37; TextOff 'Change the language / Zmiana języka / Ändere die Sprache'
      on Click: function_fb9197e8(-1)
   Button "Start screen" at 1,202 size 52x37; TextOn 'Start screen'; TextOff 'Start screen'; PictureOn "NavigateHome_KTP600_Basic_color_PN"; PictureOff "NavigateHome_KTP600_Basic_color_PN"
      on Release: ActivateScreen("Root screen", 0); SetTag("GameType", 0)
   SymbolicIOField "Template_Symbolic I/O field_1" at 15,15 size 50x50; TextOn '1'; TextOff '0'; TextList "3x3_TextList"
      ProcessValue <- "t00_HMI"
   SymbolicIOField "Template_Symbolic I/O field_2" at 75,15 size 50x50; TextOn '1'; TextOff '0'; TextList "3x3_TextList"
      ProcessValue <- "t01_HMI"
   SymbolicIOField "Template_Symbolic I/O field_3" at 135,15 size 50x50; TextOn '1'; TextOff '0'; TextList "3x3_TextList"
      ProcessValue <- "t02_HMI"
   SymbolicIOField "Template_Symbolic I/O field_4" at 15,75 size 50x50; TextOn '1'; TextOff '0'; TextList "3x3_TextList"
      ProcessValue <- "t10_HMI"
   SymbolicIOField "Template_Symbolic I/O field_5" at 75,75 size 50x50; TextOn '1'; TextOff '0'; TextList "3x3_TextList"
      ProcessValue <- "t11_HMI"
   SymbolicIOField "Template_Symbolic I/O field_6" at 135,75 size 50x50; TextOn '1'; TextOff '0'; TextList "3x3_TextList"
      ProcessValue <- "t12_HMI"
   SymbolicIOField "Template_Symbolic I/O field_7" at 15,135 size 50x50; TextOn '1'; TextOff '0'; TextList "3x3_TextList"
      ProcessValue <- "t20_HMI"
   SymbolicIOField "Template_Symbolic I/O field_8" at 75,135 size 50x50; TextOn '1'; TextOff '0'; TextList "3x3_TextList"
      ProcessValue <- "t21_HMI"
   SymbolicIOField "Template_Symbolic I/O field_9" at 135,135 size 50x50; TextOn '1'; TextOff '0'; TextList "3x3_TextList"
      ProcessValue <- "t22_HMI"

Template "4x4Template" 320x240
   Button "Exit" at 266,202 size 52x37; TextOn 'Exit'; TextOff 'Exit'; PictureOn "ExitRuntime_KTP600_Basic_color_PN"; PictureOff "ExitRuntime_KTP600_Basic_color_PN"
      on Release: StopRuntime(0)
   Button "Template_Button_3" at 54,202 size 212x37; TextOff 'Change the language / Zmiana języka / Ändere die Sprache'
      on Click: function_fb9197e8(-1)
   Button "Start screen" at 1,202 size 52x37; TextOn 'Start screen'; TextOff 'Start screen'; PictureOn "NavigateHome_KTP600_Basic_color_PN"; PictureOff "NavigateHome_KTP600_Basic_color_PN"
      on Release: ActivateScreen("Root screen", 0); SetTag("GameType", 0)
   SymbolicIOField "Template_Symbolic I/O field_1" at 15,15 size 35x35; TextOn '1'; TextOff '0'; TextList "3x3_TextList"
      ProcessValue <- "t00_HMI"
   SymbolicIOField "Template_Symbolic I/O field_2" at 60,15 size 35x35; TextOn '1'; TextOff '0'; TextList "3x3_TextList"
      ProcessValue <- "t01_HMI"
   SymbolicIOField "Template_Symbolic I/O field_3" at 105,15 size 35x35; TextOn '1'; TextOff '0'; TextList "3x3_TextList"
      ProcessValue <- "t02_HMI"
   SymbolicIOField "Template_Symbolic I/O field_4" at 15,60 size 35x35; TextOn '1'; TextOff '0'; TextList "3x3_TextList"
      ProcessValue <- "t10_HMI"
   SymbolicIOField "Template_Symbolic I/O field_5" at 60,60 size 35x35; TextOn '1'; TextOff '0'; TextList "3x3_TextList"
      ProcessValue <- "t11_HMI"
   SymbolicIOField "Template_Symbolic I/O field_6" at 105,60 size 35x35; TextOn '1'; TextOff '0'; TextList "3x3_TextList"
      ProcessValue <- "t12_HMI"
   SymbolicIOField "Template_Symbolic I/O field_7" at 15,105 size 35x35; TextOn '1'; TextOff '0'; TextList "3x3_TextList"
      ProcessValue <- "t20_HMI"
   SymbolicIOField "Template_Symbolic I/O field_8" at 60,105 size 35x35; TextOn '1'; TextOff '0'; TextList "3x3_TextList"
      ProcessValue <- "t21_HMI"
   SymbolicIOField "Template_Symbolic I/O field_9" at 105,105 size 35x35; TextOn '1'; TextOff '0'; TextList "3x3_TextList"
      ProcessValue <- "t22_HMI"
   SymbolicIOField "Template_Symbolic I/O field_10" at 15,150 size 35x35; TextOn '1'; TextOff '0'; TextList "3x3_TextList"
      ProcessValue <- "t30_HMI"
   SymbolicIOField "Template_Symbolic I/O field_11" at 60,150 size 35x35; TextOn '1'; TextOff '0'; TextList "3x3_TextList"
      ProcessValue <- "t31_HMI"
   SymbolicIOField "Template_Symbolic I/O field_12" at 105,150 size 35x35; TextOn '1'; TextOff '0'; TextList "3x3_TextList"
      ProcessValue <- "t32_HMI"
   SymbolicIOField "Template_Symbolic I/O field_13" at 150,15 size 35x35; TextOn '1'; TextOff '0'; TextList "3x3_TextList"
      ProcessValue <- "t03_HMI"
   SymbolicIOField "Template_Symbolic I/O field_14" at 150,60 size 35x35; TextOn '1'; TextOff '0'; TextList "3x3_TextList"
      ProcessValue <- "t13_HMI"
   SymbolicIOField "Template_Symbolic I/O field_15" at 150,105 size 35x35; TextOn '1'; TextOff '0'; TextList "3x3_TextList"
      ProcessValue <- "t23_HMI"
   SymbolicIOField "Template_Symbolic I/O field_16" at 150,150 size 35x35; TextOn '1'; TextOff '0'; TextList "3x3_TextList"
      ProcessValue <- "t33_HMI"

screen "4x4PvP" 320x240, template "4x4Template"
   Button "Button_3" at 15,15 size 35x35; TextOff 't00'; TextList "3x3_TextList"
      on Release: ResetBit("t00btn_HMI"); InvertBit("x")
      on Press: SetBit("t00btn_HMI")
      ProcessValue <- "t00(1)"
   Button "Button_5" at 105,15 size 35x35; TextOff 't02'; TextList "3x3_TextList"
      on Release: ResetBit("t02btn_HMI"); InvertBit("x")
      on Press: SetBit("t02btn_HMI")
      ProcessValue <- "t00(1)"
   Button "Button_1" at 60,15 size 35x35; TextOff 't01'; TextList "3x3_TextList"
      on Release: ResetBit("t01btn_HMI"); InvertBit("x")
      on Press: SetBit("t01btn_HMI")
      ProcessValue <- "t00(1)"
   Button "Button_6" at 15,60 size 35x35; TextOff 't10'; TextList "3x3_TextList"
      on Release: ResetBit("t10btn_HMI"); InvertBit("x")
      on Press: SetBit("t10btn_HMI")
      ProcessValue <- "t00(1)"
   Button "Button_7" at 105,60 size 35x35; TextOff 't12'; TextList "3x3_TextList"
      on Release: ResetBit("t12btn_HMI"); InvertBit("x")
      on Press: SetBit("t12btn_HMI")
      ProcessValue <- "t00(1)"
   Button "Button_8" at 60,60 size 35x35; TextOff 't11'; TextList "3x3_TextList"
      on Release: ResetBit("t11btn_HMI"); InvertBit("x")
      on Press: SetBit("t11btn_HMI")
      ProcessValue <- "t00(1)"
   Button "Button_9" at 15,105 size 35x35; TextOff 't20'; TextList "3x3_TextList"
      on Release: ResetBit("t20btn_HMI"); InvertBit("x")
      on Press: SetBit("t20btn_HMI")
      ProcessValue <- "t00(1)"
   Button "Button_10" at 105,105 size 35x35; TextOff 't22'; TextList "3x3_TextList"
      on Release: ResetBit("t22btn_HMI"); InvertBit("x")
      on Press: SetBit("t22btn_HMI")
      ProcessValue <- "t00(1)"
   Button "Button_11" at 60,105 size 35x35; TextOff 't21'; TextList "3x3_TextList"
      on Release: ResetBit("t21btn_HMI"); InvertBit("x")
      on Press: SetBit("t21btn_HMI")
      ProcessValue <- "t00(1)"
   Button "Button_2" at 150,15 size 35x35; TextOff 't02'; TextList "3x3_TextList"
      on Release: ResetBit("t03btn_HMI"); InvertBit("x")
      on Press: SetBit("t03btn_HMI")
      ProcessValue <- "t00(1)"
   Button "Button_4" at 150,60 size 35x35; TextOff 't12'; TextList "3x3_TextList"
      on Release: ResetBit("t13btn_HMI"); InvertBit("x")
      on Press: SetBit("t13btn_HMI")
      ProcessValue <- "t00(1)"
   Button "Button_12" at 150,105 size 35x35; TextOff 't22'; TextList "3x3_TextList"
      on Release: ResetBit("t23btn_HMI"); InvertBit("x")
      on Press: SetBit("t23btn_HMI")
      ProcessValue <- "t00(1)"
   Button "Button_13" at 15,150 size 35x35; TextOff 't20'; TextList "3x3_TextList"
      on Release: ResetBit("t30btn_HMI"); InvertBit("x")
      on Press: SetBit("t30btn_HMI")
      ProcessValue <- "t00(1)"
   Button "Button_14" at 105,150 size 35x35; TextOff 't22'; TextList "3x3_TextList"
      on Release: ResetBit("t32btn_HMI"); InvertBit("x")
      on Press: SetBit("t32btn_HMI")
      ProcessValue <- "t00(1)"
   Button "Button_15" at 60,150 size 35x35; TextOff 't21'; TextList "3x3_TextList"
      on Release: ResetBit("t31btn_HMI"); InvertBit("x")
      on Press: SetBit("t31btn_HMI")
      ProcessValue <- "t00(1)"
   Button "Button_16" at 150,150 size 35x35; TextOff 't22'; TextList "3x3_TextList"
      on Release: ResetBit("t33btn_HMI"); InvertBit("x")
      on Press: SetBit("t33btn_HMI")
      ProcessValue <- "t00(1)"
   Button "Button_17" at 220,89 size 85x85; TextOff 'Reset'
      on Release: ResetBit("Reset")
      on Press: SetBit("Reset")
   SymbolicIOField "Symbolic I/O field_1" at 220,31 size 85x44; TextOn '1'; TextOff '0'; TextList "WinInfo_TextList"
      ProcessValue <- "WinValue"

screen "4x4PvC" 320x240, template "4x4Template"
   Button "Button_17" at 220,89 size 85x85; TextOff 'Reset'
      on Release: ResetBit("Reset")
      on Press: SetBit("Reset")
   Button "Button_3" at 15,15 size 35x35; TextOff 't00'; TextList "3x3_TextList"
      on Release: ResetBit("t00btn_HMI"); InvertBit("x")
      on Press: SetBit("t00btn_HMI")
      ProcessValue <- "t00(1)"
   Button "Button_5" at 105,15 size 35x35; TextOff 't02'; TextList "3x3_TextList"
      on Release: ResetBit("t02btn_HMI"); InvertBit("x")
      on Press: SetBit("t02btn_HMI")
      ProcessValue <- "t00(1)"
   Button "Button_1" at 60,15 size 35x35; TextOff 't01'; TextList "3x3_TextList"
      on Release: ResetBit("t01btn_HMI"); InvertBit("x")
      on Press: SetBit("t01btn_HMI")
      ProcessValue <- "t00(1)"
   Button "Button_6" at 15,60 size 35x35; TextOff 't10'; TextList "3x3_TextList"
      on Release: ResetBit("t10btn_HMI"); InvertBit("x")
      on Press: SetBit("t10btn_HMI")
      ProcessValue <- "t00(1)"
   Button "Button_7" at 105,60 size 35x35; TextOff 't12'; TextList "3x3_TextList"
      on Release: ResetBit("t12btn_HMI"); InvertBit("x")
      on Press: SetBit("t12btn_HMI")
      ProcessValue <- "t00(1)"
   Button "Button_8" at 60,60 size 35x35; TextOff 't11'; TextList "3x3_TextList"
      on Release: ResetBit("t11btn_HMI"); InvertBit("x")
      on Press: SetBit("t11btn_HMI")
      ProcessValue <- "t00(1)"
   Button "Button_9" at 15,105 size 35x35; TextOff 't20'; TextList "3x3_TextList"
      on Release: ResetBit("t20btn_HMI"); InvertBit("x")
      on Press: SetBit("t20btn_HMI")
      ProcessValue <- "t00(1)"
   Button "Button_10" at 105,105 size 35x35; TextOff 't22'; TextList "3x3_TextList"
      on Release: ResetBit("t22btn_HMI"); InvertBit("x")
      on Press: SetBit("t22btn_HMI")
      ProcessValue <- "t00(1)"
   Button "Button_11" at 60,105 size 35x35; TextOff 't21'; TextList "3x3_TextList"
      on Release: ResetBit("t21btn_HMI"); InvertBit("x")
      on Press: SetBit("t21btn_HMI")
      ProcessValue <- "t00(1)"
   Button "Button_2" at 150,15 size 35x35; TextOff 't02'; TextList "3x3_TextList"
      on Release: ResetBit("t03btn_HMI"); InvertBit("x")
      on Press: SetBit("t03btn_HMI")
      ProcessValue <- "t00(1)"
   Button "Button_4" at 150,60 size 35x35; TextOff 't12'; TextList "3x3_TextList"
      on Release: ResetBit("t13btn_HMI"); InvertBit("x")
      on Press: SetBit("t13btn_HMI")
      ProcessValue <- "t00(1)"
   Button "Button_12" at 150,105 size 35x35; TextOff 't22'; TextList "3x3_TextList"
      on Release: ResetBit("t23btn_HMI"); InvertBit("x")
      on Press: SetBit("t23btn_HMI")
      ProcessValue <- "t00(1)"
   Button "Button_13" at 15,150 size 35x35; TextOff 't20'; TextList "3x3_TextList"
      on Release: ResetBit("t30btn_HMI"); InvertBit("x")
      on Press: SetBit("t30btn_HMI")
      ProcessValue <- "t00(1)"
   Button "Button_14" at 105,150 size 35x35; TextOff 't22'; TextList "3x3_TextList"
      on Release: ResetBit("t32btn_HMI"); InvertBit("x")
      on Press: SetBit("t32btn_HMI")
      ProcessValue <- "t00(1)"
   Button "Button_15" at 60,150 size 35x35; TextOff 't21'; TextList "3x3_TextList"
      on Release: ResetBit("t31btn_HMI"); InvertBit("x")
      on Press: SetBit("t31btn_HMI")
      ProcessValue <- "t00(1)"
   Button "Button_16" at 150,150 size 35x35; TextOff 't22'; TextList "3x3_TextList"
      on Release: ResetBit("t33btn_HMI"); InvertBit("x")
      on Press: SetBit("t33btn_HMI")
      ProcessValue <- "t00(1)"
   SymbolicIOField "Symbolic I/O field_1" at 220,31 size 85x44; TextOn '1'; TextOff '0'; TextList "WinInfo_TextList"
      ProcessValue <- "WinValue"
*)